// TIA Portal V16 export
// export: Created 2020-03-17T19:47:24.6378532Z, ExportSetting None, DisplayName Totally Integrated Automation Portal, DisplayVersion V16, DisplayName TIA Portal Version Control Interface, DisplayVersion V16, DisplayName TIA Portal Openness, DisplayVersion V16, DisplayName STEP 7 Professional, DisplayVersion V16, DisplayName STEP 7 Safety, DisplayVersion V16, DisplayName WinCC Advanced, DisplayVersion V16
FUNCTION_BLOCK "FB_R134a_BU_Valves"   // FB1303, LAD
TITLE = Base unit valve control // Grundeinheit Ventilsteuerung
{ S7_Optimized_Access := 'TRUE' }
// stored: AutoNumber false, MemoryReserve 100, SetENOAutomatically false
   VAR
      Stat_Flag : Array[1..32] of Bool;   // Bits for edge detection // Bits für Flankenerkennung
      Valve_10 : "FB_VALVE";
      Valve_12 : "FB_VALVE";
      Valve_13 : "FB_VALVE";
      Valve_16 : "FB_VALVE";
      Valve_17 : "FB_VALVE";
      Valve_18 : "FB_VALVE";
      Valve_19 : "FB_VALVE";
      Valve_20 : "FB_VALVE";
      Valve_21 : "FB_VALVE";
      Valve_23 : "FB_VALVE";
      Valve_24 : "FB_VALVE";
      Valve_31 : "FB_VALVE";
      Valve_43 : "FB_VALVE";
      Valve_44 : "FB_VALVE";
      Valve_Spare_1 : "FB_VALVE";
      Valve_Spare_2 : "FB_VALVE";
      Valve_Spare_3 : "FB_VALVE";
      Valve_Spare_4 : "FB_VALVE";
      Valve_Spare_5 : "FB_VALVE";
      Valve_Spare_6 : "FB_VALVE";
   END_VAR
   VAR_TEMP
      Tmp_EnableMonitoring : Bool;   // Local monitoring release // Lokale Überwachungsfreigabe
      Tmp_EnableOperation : Bool;   // Local operation release // Lokale Startfreigabe
      Tmp_Bool : Bool;   // Placeholder BOOL // Platzhalter BOOL
      Tmp_Word : Word;   // Placeholder WORD // Platzhalter WORD
      Tmp_Int : Int;   // Placeholder INT // Platzhalter INT
      Tmp_Alarm : Array[1..4] of Bool;   // Temp variable for FB_Alarm // Temporäre Variablen für den FB_Alarm
      Tmp_CollectedAlarm : Bool;   // Temp collected alarm for FB_Alarm // Temporärer Sammelfehler für FB_Alarm
      Tmp_OffsetPropValveAir : Int;   // Offset value for proportional valve // Offsetwert für Proportionalventil
      Tmp_OffsetPropValveFluid : Int;   // Offset value for proportional valve // Offsetwert für Proportionalventil
      Tmp_Fault : Bool;   // Temp variable for fault // Temporäre Variable für Fehler
      Tmp_BypassRelivePressure : Bool;   // Bypass for function relive pressure // Beipass für die Funktion Druck entlasten
      Tmp_ReturnValue : Word;   // Return value from function // Rückgabewert von Funktion
   END_VAR
   VAR_TEMP   // added for the SCL form of the ladder/FBD networks
      _w1 : Bool;
   END_VAR
BEGIN

REGION Network 1: Enable Monitoring // Freigabe Überwachung
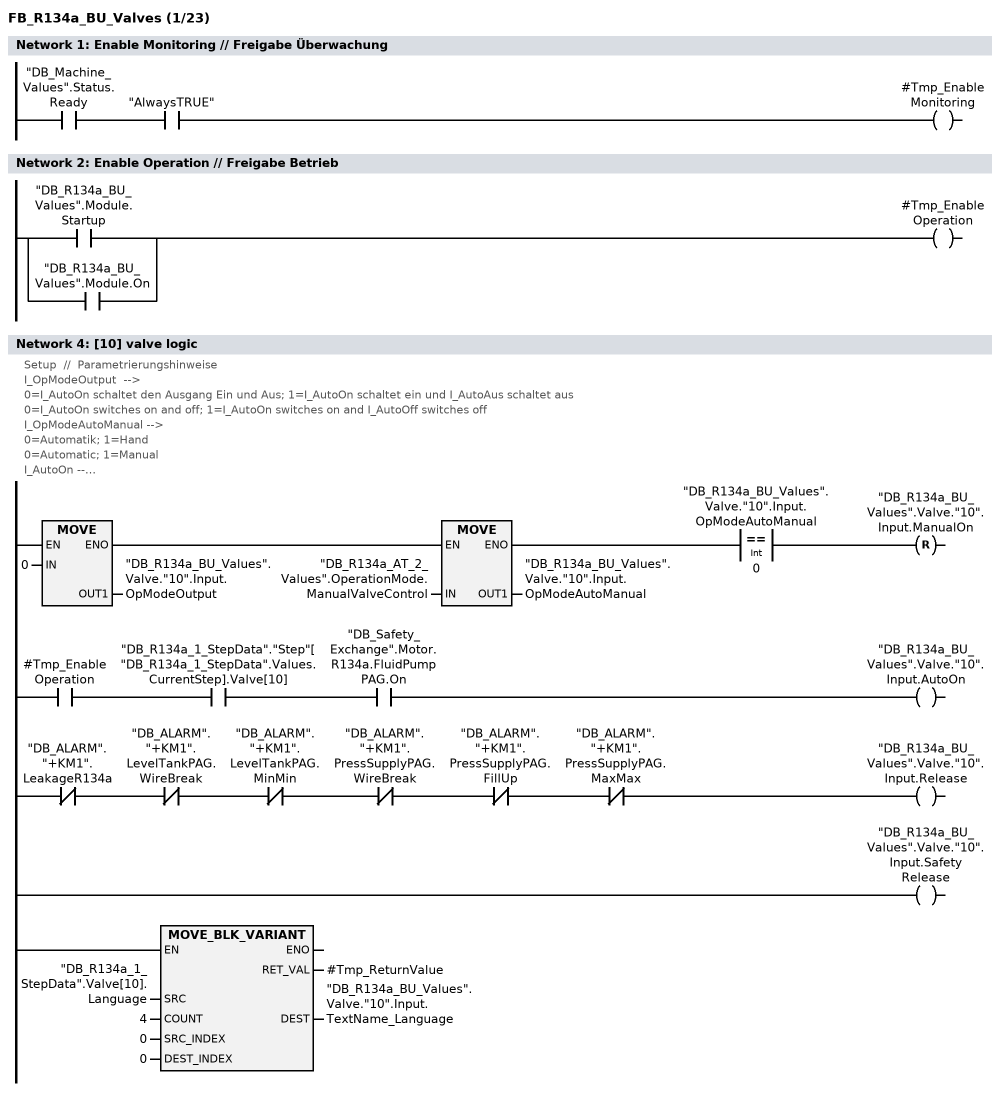
   RUNG wire#powerrail
      Contact( "DB_Machine_Values".Status.Ready )
      Contact( "AlwaysTRUE" )
      Coil( #Tmp_EnableMonitoring )
   END_RUNG
   // the same network as SCL:
   #Tmp_EnableMonitoring := "DB_Machine_Values".Status.Ready AND "AlwaysTRUE";
END_REGION

REGION Network 2: Enable Operation // Freigabe Betrieb
   RUNG wire#powerrail
      Contact( "DB_R134a_BU_Values".Module.Startup )
      wire#w1
      Coil( #Tmp_EnableOperation )
   END_RUNG
   RUNG wire#powerrail
      Contact( "DB_R134a_BU_Values".Module.On )
   END_RUNG wire#w1
   // the same network as SCL:
   #Tmp_EnableOperation := "DB_R134a_BU_Values".Module.Startup OR "DB_R134a_BU_Values".Module.On;
END_REGION

REGION Network 3: ------------- Valves base unit -------------
   // This network is only here to make the PLC program more structured/readable // Dieses Netzwerk ist nur hier um die Lesbarkeit des SPS-Programms zu erhöhen
END_REGION

REGION Network 4: [10] valve logic
   // Setup  //  Parametrierungshinweise
   // I_OpModeOutput  -->
   // 0=I_AutoOn schaltet den Ausgang Ein und Aus; 1=I_AutoOn schaltet ein und I_AutoAus schaltet aus
   // 0=I_AutoOn switches on and off; 1=I_AutoOn switches on and I_AutoOff switches off
   // 
   // I_OpModeAutoManual -->
   // 0=Automatik; 1=Hand
   // 0=Automatic; 1=Manual
   // 
   // I_AutoOn -->
   // 1=Automatik Ein, Eingang für die normalen Ventilverschaltungsbedingungen
   // 1=Automatic On, Input for the normal valve conditions
   // 
   // I_Release -->
   // 1=Freigabe, Eingang für die Fehlerbedingungen
   // 1=Release, Input for fault conditions
   // 
   // I_SafetyRelease -->
   // 1=Sicherheitsfreigabe, Eingang für zusätzliche Schaltbefehle aus dem Sicherheitsprogramm
   // 1=Safety release, Input for additional safety conditions from the safety program
   RUNG wire#powerrail
      Move(in := 0, out1 => "DB_R134a_BU_Values".Valve."10".Input.OpModeOutput)
      Move(in := "DB_R134a_AT_2_Values".OperationMode.ManualValveControl, out1 => "DB_R134a_BU_Values".Valve."10".Input.OpModeAutoManual)
      { S7_Templates := "SrcType := Int" } EQ_Contact(in1 := "DB_R134a_BU_Values".Valve."10".Input.OpModeAutoManual, in2 := 0)
      R_Coil( "DB_R134a_BU_Values".Valve."10".Input.ManualOn )
   END_RUNG
   RUNG wire#powerrail
      Contact( #Tmp_EnableOperation )
      Contact( "DB_R134a_1_StepData"."Step"["DB_R134a_1_StepData".Values.CurrentStep].Valve[10] )
      Contact( "DB_Safety_Exchange".Motor.R134a.FluidPumpPAG.On )
      Coil( "DB_R134a_BU_Values".Valve."10".Input.AutoOn )
   END_RUNG
   RUNG wire#powerrail
      I_Contact( "DB_ALARM"."+KM1".LeakageR134a )
      I_Contact( "DB_ALARM"."+KM1".LevelTankPAG.WireBreak )
      I_Contact( "DB_ALARM"."+KM1".LevelTankPAG.MinMin )
      I_Contact( "DB_ALARM"."+KM1".PressSupplyPAG.WireBreak )
      I_Contact( "DB_ALARM"."+KM1".PressSupplyPAG.FillUp )
      I_Contact( "DB_ALARM"."+KM1".PressSupplyPAG.MaxMax )
      Coil( "DB_R134a_BU_Values".Valve."10".Input.Release )
   END_RUNG
   RUNG wire#powerrail
      Coil( "DB_R134a_BU_Values".Valve."10".Input.SafetyRelease )
   END_RUNG
   RUNG wire#powerrail
      MOVE_BLK_VARIANT(SRC := "DB_R134a_1_StepData".Valve[10].Language, COUNT := 4, SRC_INDEX := 0, DEST_INDEX := 0, Ret_Val => #Tmp_ReturnValue, DEST => "DB_R134a_BU_Values".Valve."10".Input.TextName_Language)
   END_RUNG
   // the same network as SCL:
   "DB_R134a_BU_Values".Valve."10".Input.OpModeOutput := 0;
   "DB_R134a_BU_Values".Valve."10".Input.OpModeAutoManual := "DB_R134a_AT_2_Values".OperationMode.ManualValveControl;
   IF "DB_R134a_BU_Values".Valve."10".Input.OpModeAutoManual = 0 THEN
       "DB_R134a_BU_Values".Valve."10".Input.ManualOn := FALSE;
   END_IF;
   "DB_R134a_BU_Values".Valve."10".Input.AutoOn := #Tmp_EnableOperation AND "DB_R134a_1_StepData"."Step"["DB_R134a_1_StepData".Values.CurrentStep].Valve[10] AND "DB_Safety_Exchange".Motor.R134a.FluidPumpPAG.On;
   "DB_R134a_BU_Values".Valve."10".Input.Release := NOT "DB_ALARM"."+KM1".LeakageR134a AND NOT "DB_ALARM"."+KM1".LevelTankPAG.WireBreak AND NOT "DB_ALARM"."+KM1".LevelTankPAG.MinMin AND NOT "DB_ALARM"."+KM1".PressSupplyPAG.WireBreak AND NOT "DB_ALARM"."+KM1".PressSupplyPAG.FillUp AND NOT "DB_ALARM"."+KM1".PressSupplyPAG.MaxMax;
   "DB_R134a_BU_Values".Valve."10".Input.SafetyRelease := TRUE;
   #Tmp_ReturnValue := MOVE_BLK_VARIANT(SRC := "DB_R134a_1_StepData".Valve[10].Language,
                           COUNT := 4,
                           SRC_INDEX := 0,
                           DEST_INDEX := 0,
                           DEST => "DB_R134a_BU_Values".Valve."10".Input.TextName_Language);
END_REGION

REGION Network 5: [10] valve 1KM1VI1KKP9KK101 - 100.101.6 - Charge accumulator PAG // Füllen PAG-Speicher
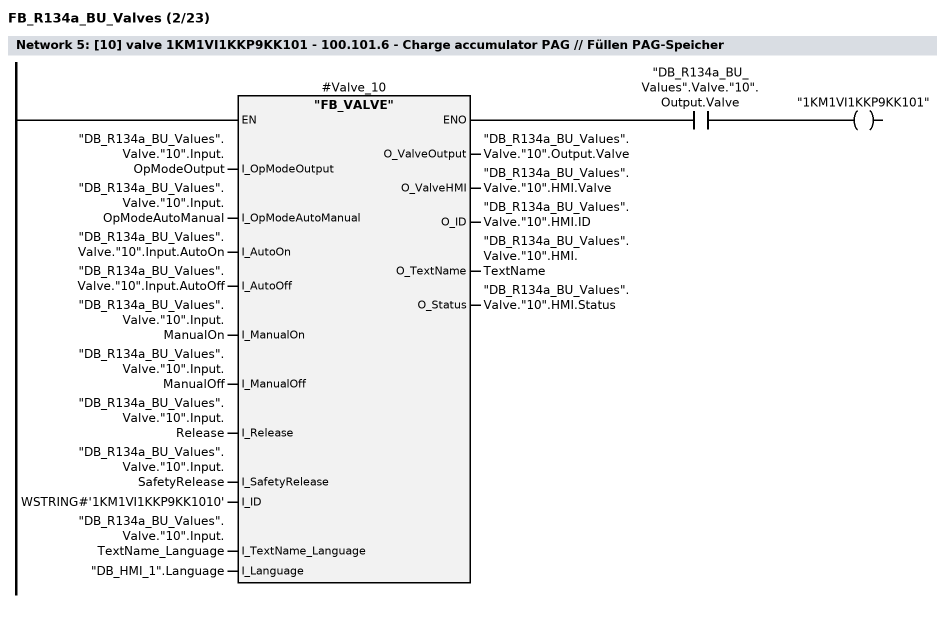
   RUNG wire#powerrail
      #Valve_10(I_OpModeOutput := "DB_R134a_BU_Values".Valve."10".Input.OpModeOutput, I_OpModeAutoManual := "DB_R134a_BU_Values".Valve."10".Input.OpModeAutoManual, I_AutoOn := "DB_R134a_BU_Values".Valve."10".Input.AutoOn, I_AutoOff := "DB_R134a_BU_Values".Valve."10".Input.AutoOff, I_ManualOn := "DB_R134a_BU_Values".Valve."10".Input.ManualOn, I_ManualOff := "DB_R134a_BU_Values".Valve."10".Input.ManualOff, I_Release := "DB_R134a_BU_Values".Valve."10".Input.Release, I_SafetyRelease := "DB_R134a_BU_Values".Valve."10".Input.SafetyRelease, I_ID := WSTRING#'1KM1VI1KKP9KK1010', I_TextName_Language := "DB_R134a_BU_Values".Valve."10".Input.TextName_Language, I_Language := "DB_HMI_1".Language, O_ValveOutput => "DB_R134a_BU_Values".Valve."10".Output.Valve, O_ValveHMI => "DB_R134a_BU_Values".Valve."10".HMI.Valve, O_ID => "DB_R134a_BU_Values".Valve."10".HMI.ID, O_TextName => "DB_R134a_BU_Values".Valve."10".HMI.TextName, O_Status => "DB_R134a_BU_Values".Valve."10".HMI.Status)
      Contact( "DB_R134a_BU_Values".Valve."10".Output.Valve )
      Coil( "1KM1VI1KKP9KK101" )
   END_RUNG
   // the same network as SCL:
   #Valve_10(I_OpModeOutput := "DB_R134a_BU_Values".Valve."10".Input.OpModeOutput,   // "FB_VALVE"
             I_OpModeAutoManual := "DB_R134a_BU_Values".Valve."10".Input.OpModeAutoManual,
             I_AutoOn := "DB_R134a_BU_Values".Valve."10".Input.AutoOn,
             I_AutoOff := "DB_R134a_BU_Values".Valve."10".Input.AutoOff,
             I_ManualOn := "DB_R134a_BU_Values".Valve."10".Input.ManualOn,
             I_ManualOff := "DB_R134a_BU_Values".Valve."10".Input.ManualOff,
             I_Release := "DB_R134a_BU_Values".Valve."10".Input.Release,
             I_SafetyRelease := "DB_R134a_BU_Values".Valve."10".Input.SafetyRelease,
             I_ID := WSTRING#'1KM1VI1KKP9KK1010',
             I_TextName_Language := "DB_R134a_BU_Values".Valve."10".Input.TextName_Language,
             I_Language := "DB_HMI_1".Language,
             O_ValveOutput => "DB_R134a_BU_Values".Valve."10".Output.Valve,
             O_ValveHMI => "DB_R134a_BU_Values".Valve."10".HMI.Valve,
             O_ID => "DB_R134a_BU_Values".Valve."10".HMI.ID,
             O_TextName => "DB_R134a_BU_Values".Valve."10".HMI.TextName,
             O_Status => "DB_R134a_BU_Values".Valve."10".HMI.Status,
             ENO => #_w1);
   "1KM1VI1KKP9KK101" := #_w1 AND "DB_R134a_BU_Values".Valve."10".Output.Valve;
END_REGION

REGION Network 6: [12] valve logic
   // Setup  //  Parametrierungshinweise
   // I_OpModeOutput  -->
   // 0=I_AutoOn schaltet den Ausgang Ein und Aus; 1=I_AutoOn schaltet ein und I_AutoAus schaltet aus
   // 0=I_AutoOn switches on and off; 1=I_AutoOn switches on and I_AutoOff switches off
   // 
   // I_OpModeAutoManual -->
   // 0=Automatik; 1=Hand
   // 0=Automatic; 1=Manual
   // 
   // I_AutoOn -->
   // 1=Automatik Ein, Eingang für die normalen Ventilverschaltungsbedingungen
   // 1=Automatic On, Input for the normal valve conditions
   // 
   // I_Release -->
   // 1=Freigabe, Eingang für die Fehlerbedingungen
   // 1=Release, Input for fault conditions
   // 
   // I_SafetyRelease -->
   // 1=Sicherheitsfreigabe, Eingang für zusätzliche Schaltbefehle aus dem Sicherheitsprogramm
   // 1=Safety release, Input for additional safety conditions from the safety program
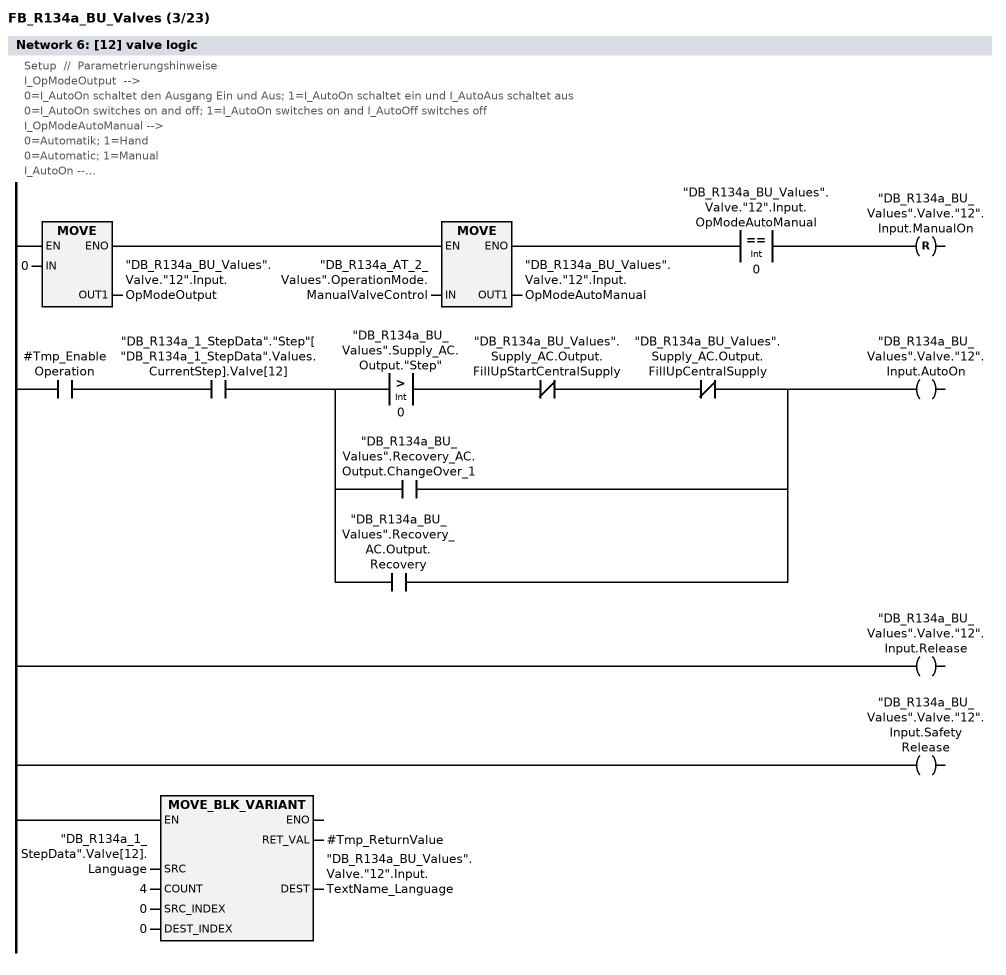
   RUNG wire#powerrail
      Move(in := 0, out1 => "DB_R134a_BU_Values".Valve."12".Input.OpModeOutput)
      Move(in := "DB_R134a_AT_2_Values".OperationMode.ManualValveControl, out1 => "DB_R134a_BU_Values".Valve."12".Input.OpModeAutoManual)
      { S7_Templates := "SrcType := Int" } EQ_Contact(in1 := "DB_R134a_BU_Values".Valve."12".Input.OpModeAutoManual, in2 := 0)
      R_Coil( "DB_R134a_BU_Values".Valve."12".Input.ManualOn )
   END_RUNG
   RUNG wire#powerrail
      Contact( #Tmp_EnableOperation )
      Contact( "DB_R134a_1_StepData"."Step"["DB_R134a_1_StepData".Values.CurrentStep].Valve[12] )
      wire#w1
      { S7_Templates := "SrcType := Int" } GT_Contact(in1 := "DB_R134a_BU_Values".Supply_AC.Output."Step", in2 := 0)
      I_Contact( "DB_R134a_BU_Values".Supply_AC.Output.FillUpStartCentralSupply )
      I_Contact( "DB_R134a_BU_Values".Supply_AC.Output.FillUpCentralSupply )
      wire#w2
      Coil( "DB_R134a_BU_Values".Valve."12".Input.AutoOn )
   END_RUNG
   RUNG wire#w1
      Contact( "DB_R134a_BU_Values".Recovery_AC.Output.ChangeOver_1 )
   END_RUNG wire#w2
   RUNG wire#w1
      Contact( "DB_R134a_BU_Values".Recovery_AC.Output.Recovery )
   END_RUNG wire#w2
   RUNG wire#powerrail
      Coil( "DB_R134a_BU_Values".Valve."12".Input.Release )
   END_RUNG
   RUNG wire#powerrail
      Coil( "DB_R134a_BU_Values".Valve."12".Input.SafetyRelease )
   END_RUNG
   RUNG wire#powerrail
      MOVE_BLK_VARIANT(SRC := "DB_R134a_1_StepData".Valve[12].Language, COUNT := 4, SRC_INDEX := 0, DEST_INDEX := 0, Ret_Val => #Tmp_ReturnValue, DEST => "DB_R134a_BU_Values".Valve."12".Input.TextName_Language)
   END_RUNG
   // the same network as SCL:
   "DB_R134a_BU_Values".Valve."12".Input.OpModeOutput := 0;
   "DB_R134a_BU_Values".Valve."12".Input.OpModeAutoManual := "DB_R134a_AT_2_Values".OperationMode.ManualValveControl;
   IF "DB_R134a_BU_Values".Valve."12".Input.OpModeAutoManual = 0 THEN
       "DB_R134a_BU_Values".Valve."12".Input.ManualOn := FALSE;
   END_IF;
   "DB_R134a_BU_Values".Valve."12".Input.AutoOn := #Tmp_EnableOperation AND "DB_R134a_1_StepData"."Step"["DB_R134a_1_StepData".Values.CurrentStep].Valve[12] AND ((("DB_R134a_BU_Values".Supply_AC.Output."Step" > 0) AND NOT "DB_R134a_BU_Values".Supply_AC.Output.FillUpStartCentralSupply AND NOT "DB_R134a_BU_Values".Supply_AC.Output.FillUpCentralSupply) OR "DB_R134a_BU_Values".Recovery_AC.Output.ChangeOver_1 OR "DB_R134a_BU_Values".Recovery_AC.Output.Recovery);
   "DB_R134a_BU_Values".Valve."12".Input.Release := TRUE;
   "DB_R134a_BU_Values".Valve."12".Input.SafetyRelease := TRUE;
   #Tmp_ReturnValue := MOVE_BLK_VARIANT(SRC := "DB_R134a_1_StepData".Valve[12].Language,
                           COUNT := 4,
                           SRC_INDEX := 0,
                           DEST_INDEX := 0,
                           DEST => "DB_R134a_BU_Values".Valve."12".Input.TextName_Language);
END_REGION

REGION Network 7: [12] valve 1KM1VI1KKP5KK420 - 109.420.3 - Compressed air supply (pump) // Druckluft Pumpe
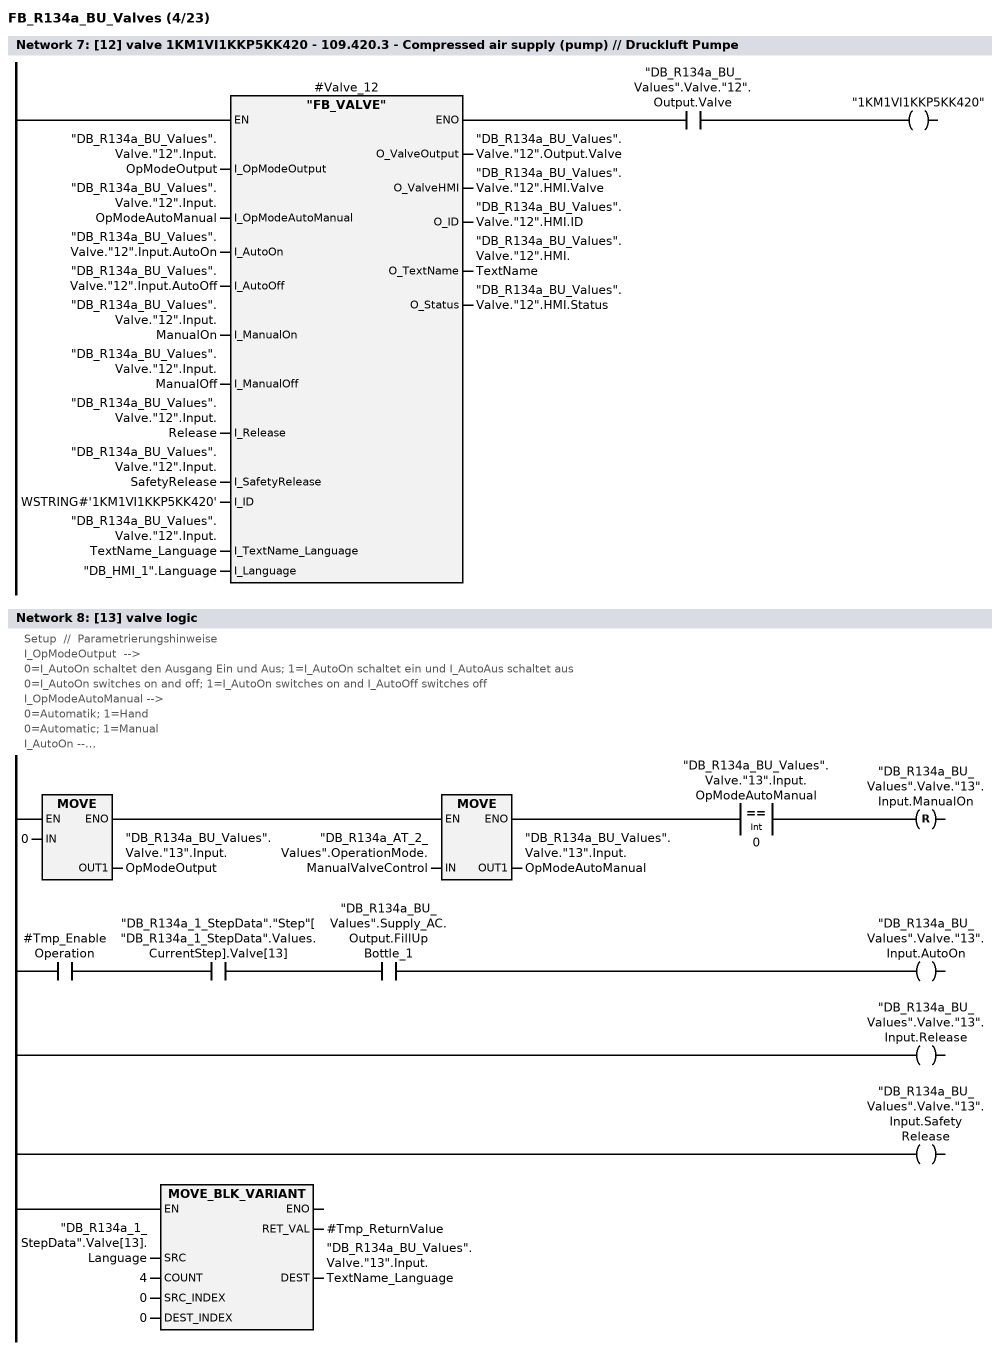
   RUNG wire#powerrail
      #Valve_12(I_OpModeOutput := "DB_R134a_BU_Values".Valve."12".Input.OpModeOutput, I_OpModeAutoManual := "DB_R134a_BU_Values".Valve."12".Input.OpModeAutoManual, I_AutoOn := "DB_R134a_BU_Values".Valve."12".Input.AutoOn, I_AutoOff := "DB_R134a_BU_Values".Valve."12".Input.AutoOff, I_ManualOn := "DB_R134a_BU_Values".Valve."12".Input.ManualOn, I_ManualOff := "DB_R134a_BU_Values".Valve."12".Input.ManualOff, I_Release := "DB_R134a_BU_Values".Valve."12".Input.Release, I_SafetyRelease := "DB_R134a_BU_Values".Valve."12".Input.SafetyRelease, I_ID := WSTRING#'1KM1VI1KKP5KK420', I_TextName_Language := "DB_R134a_BU_Values".Valve."12".Input.TextName_Language, I_Language := "DB_HMI_1".Language, O_ValveOutput => "DB_R134a_BU_Values".Valve."12".Output.Valve, O_ValveHMI => "DB_R134a_BU_Values".Valve."12".HMI.Valve, O_ID => "DB_R134a_BU_Values".Valve."12".HMI.ID, O_TextName => "DB_R134a_BU_Values".Valve."12".HMI.TextName, O_Status => "DB_R134a_BU_Values".Valve."12".HMI.Status)
      Contact( "DB_R134a_BU_Values".Valve."12".Output.Valve )
      Coil( "1KM1VI1KKP5KK420" )
   END_RUNG
   // the same network as SCL:
   #Valve_12(I_OpModeOutput := "DB_R134a_BU_Values".Valve."12".Input.OpModeOutput,   // "FB_VALVE"
             I_OpModeAutoManual := "DB_R134a_BU_Values".Valve."12".Input.OpModeAutoManual,
             I_AutoOn := "DB_R134a_BU_Values".Valve."12".Input.AutoOn,
             I_AutoOff := "DB_R134a_BU_Values".Valve."12".Input.AutoOff,
             I_ManualOn := "DB_R134a_BU_Values".Valve."12".Input.ManualOn,
             I_ManualOff := "DB_R134a_BU_Values".Valve."12".Input.ManualOff,
             I_Release := "DB_R134a_BU_Values".Valve."12".Input.Release,
             I_SafetyRelease := "DB_R134a_BU_Values".Valve."12".Input.SafetyRelease,
             I_ID := WSTRING#'1KM1VI1KKP5KK420',
             I_TextName_Language := "DB_R134a_BU_Values".Valve."12".Input.TextName_Language,
             I_Language := "DB_HMI_1".Language,
             O_ValveOutput => "DB_R134a_BU_Values".Valve."12".Output.Valve,
             O_ValveHMI => "DB_R134a_BU_Values".Valve."12".HMI.Valve,
             O_ID => "DB_R134a_BU_Values".Valve."12".HMI.ID,
             O_TextName => "DB_R134a_BU_Values".Valve."12".HMI.TextName,
             O_Status => "DB_R134a_BU_Values".Valve."12".HMI.Status,
             ENO => #_w1);
   "1KM1VI1KKP5KK420" := #_w1 AND "DB_R134a_BU_Values".Valve."12".Output.Valve;
END_REGION

REGION Network 8: [13] valve logic
   // Setup  //  Parametrierungshinweise
   // I_OpModeOutput  -->
   // 0=I_AutoOn schaltet den Ausgang Ein und Aus; 1=I_AutoOn schaltet ein und I_AutoAus schaltet aus
   // 0=I_AutoOn switches on and off; 1=I_AutoOn switches on and I_AutoOff switches off
   // 
   // I_OpModeAutoManual -->
   // 0=Automatik; 1=Hand
   // 0=Automatic; 1=Manual
   // 
   // I_AutoOn -->
   // 1=Automatik Ein, Eingang für die normalen Ventilverschaltungsbedingungen
   // 1=Automatic On, Input for the normal valve conditions
   // 
   // I_Release -->
   // 1=Freigabe, Eingang für die Fehlerbedingungen
   // 1=Release, Input for fault conditions
   // 
   // I_SafetyRelease -->
   // 1=Sicherheitsfreigabe, Eingang für zusätzliche Schaltbefehle aus dem Sicherheitsprogramm
   // 1=Safety release, Input for additional safety conditions from the safety program
   RUNG wire#powerrail
      Move(in := 0, out1 => "DB_R134a_BU_Values".Valve."13".Input.OpModeOutput)
      Move(in := "DB_R134a_AT_2_Values".OperationMode.ManualValveControl, out1 => "DB_R134a_BU_Values".Valve."13".Input.OpModeAutoManual)
      { S7_Templates := "SrcType := Int" } EQ_Contact(in1 := "DB_R134a_BU_Values".Valve."13".Input.OpModeAutoManual, in2 := 0)
      R_Coil( "DB_R134a_BU_Values".Valve."13".Input.ManualOn )
   END_RUNG
   RUNG wire#powerrail
      Contact( #Tmp_EnableOperation )
      Contact( "DB_R134a_1_StepData"."Step"["DB_R134a_1_StepData".Values.CurrentStep].Valve[13] )
      Contact( "DB_R134a_BU_Values".Supply_AC.Output.FillUpBottle_1 )
      Coil( "DB_R134a_BU_Values".Valve."13".Input.AutoOn )
   END_RUNG
   RUNG wire#powerrail
      Coil( "DB_R134a_BU_Values".Valve."13".Input.Release )
   END_RUNG
   RUNG wire#powerrail
      Coil( "DB_R134a_BU_Values".Valve."13".Input.SafetyRelease )
   END_RUNG
   RUNG wire#powerrail
      MOVE_BLK_VARIANT(SRC := "DB_R134a_1_StepData".Valve[13].Language, COUNT := 4, SRC_INDEX := 0, DEST_INDEX := 0, Ret_Val => #Tmp_ReturnValue, DEST => "DB_R134a_BU_Values".Valve."13".Input.TextName_Language)
   END_RUNG
   // the same network as SCL:
   "DB_R134a_BU_Values".Valve."13".Input.OpModeOutput := 0;
   "DB_R134a_BU_Values".Valve."13".Input.OpModeAutoManual := "DB_R134a_AT_2_Values".OperationMode.ManualValveControl;
   IF "DB_R134a_BU_Values".Valve."13".Input.OpModeAutoManual = 0 THEN
       "DB_R134a_BU_Values".Valve."13".Input.ManualOn := FALSE;
   END_IF;
   "DB_R134a_BU_Values".Valve."13".Input.AutoOn := #Tmp_EnableOperation AND "DB_R134a_1_StepData"."Step"["DB_R134a_1_StepData".Values.CurrentStep].Valve[13] AND "DB_R134a_BU_Values".Supply_AC.Output.FillUpBottle_1;
   "DB_R134a_BU_Values".Valve."13".Input.Release := TRUE;
   "DB_R134a_BU_Values".Valve."13".Input.SafetyRelease := TRUE;
   #Tmp_ReturnValue := MOVE_BLK_VARIANT(SRC := "DB_R134a_1_StepData".Valve[13].Language,
                           COUNT := 4,
                           SRC_INDEX := 0,
                           DEST_INDEX := 0,
                           DEST => "DB_R134a_BU_Values".Valve."13".Input.TextName_Language);
END_REGION

REGION Network 9: [13] valve 1KM1VI1KKP3KK30 - 100.30.3 - Supply – Bottle 1 // Versorgung - Flasche 1
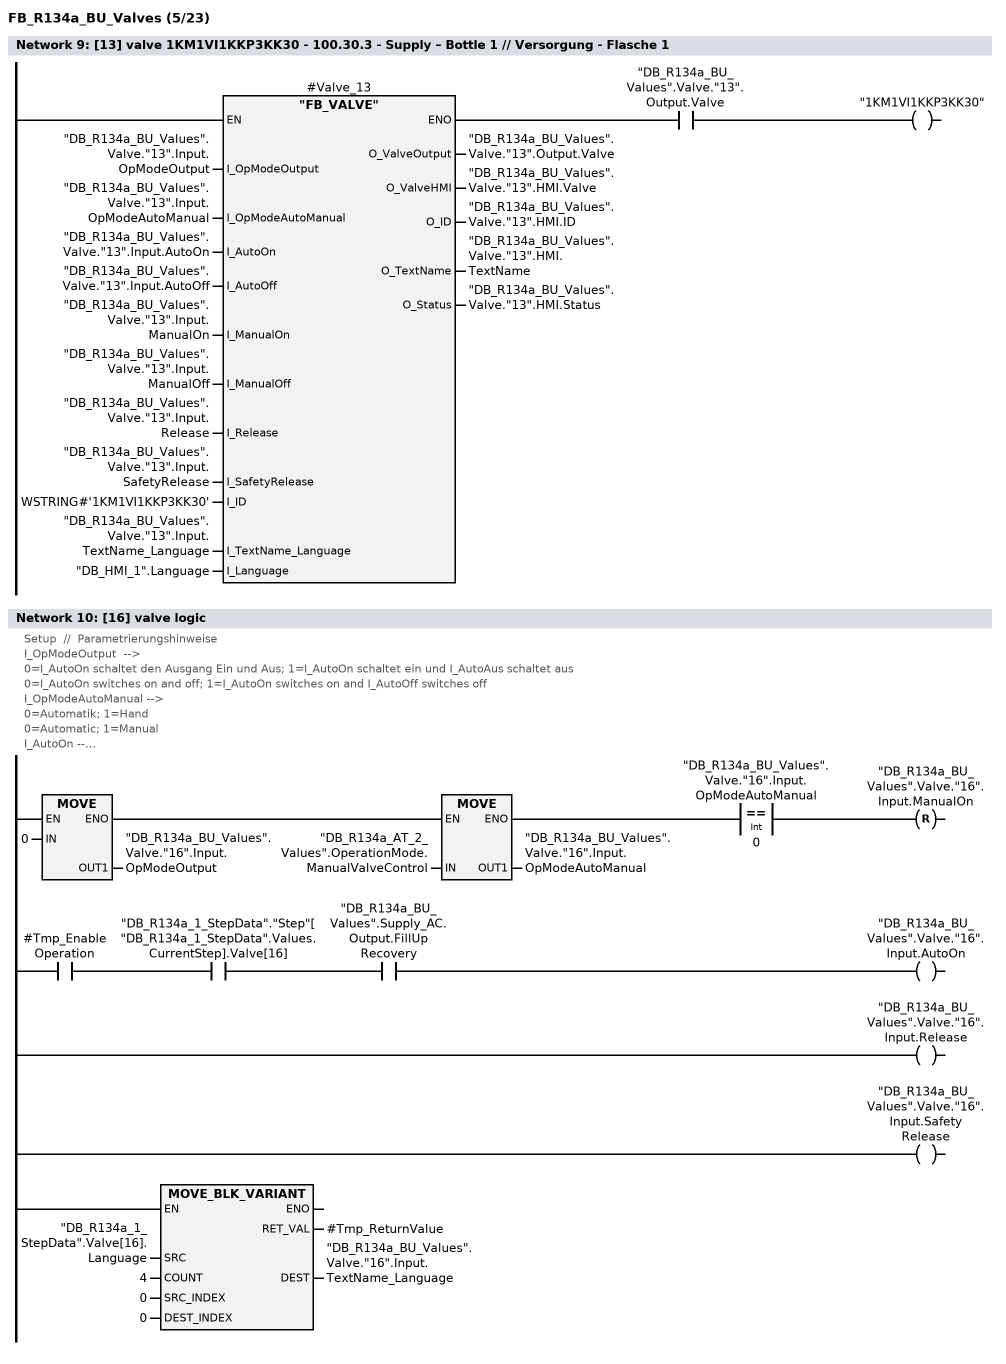
   RUNG wire#powerrail
      #Valve_13(I_OpModeOutput := "DB_R134a_BU_Values".Valve."13".Input.OpModeOutput, I_OpModeAutoManual := "DB_R134a_BU_Values".Valve."13".Input.OpModeAutoManual, I_AutoOn := "DB_R134a_BU_Values".Valve."13".Input.AutoOn, I_AutoOff := "DB_R134a_BU_Values".Valve."13".Input.AutoOff, I_ManualOn := "DB_R134a_BU_Values".Valve."13".Input.ManualOn, I_ManualOff := "DB_R134a_BU_Values".Valve."13".Input.ManualOff, I_Release := "DB_R134a_BU_Values".Valve."13".Input.Release, I_SafetyRelease := "DB_R134a_BU_Values".Valve."13".Input.SafetyRelease, I_ID := WSTRING#'1KM1VI1KKP3KK30', I_TextName_Language := "DB_R134a_BU_Values".Valve."13".Input.TextName_Language, I_Language := "DB_HMI_1".Language, O_ValveOutput => "DB_R134a_BU_Values".Valve."13".Output.Valve, O_ValveHMI => "DB_R134a_BU_Values".Valve."13".HMI.Valve, O_ID => "DB_R134a_BU_Values".Valve."13".HMI.ID, O_TextName => "DB_R134a_BU_Values".Valve."13".HMI.TextName, O_Status => "DB_R134a_BU_Values".Valve."13".HMI.Status)
      Contact( "DB_R134a_BU_Values".Valve."13".Output.Valve )
      Coil( "1KM1VI1KKP3KK30" )
   END_RUNG
   // the same network as SCL:
   #Valve_13(I_OpModeOutput := "DB_R134a_BU_Values".Valve."13".Input.OpModeOutput,   // "FB_VALVE"
             I_OpModeAutoManual := "DB_R134a_BU_Values".Valve."13".Input.OpModeAutoManual,
             I_AutoOn := "DB_R134a_BU_Values".Valve."13".Input.AutoOn,
             I_AutoOff := "DB_R134a_BU_Values".Valve."13".Input.AutoOff,
             I_ManualOn := "DB_R134a_BU_Values".Valve."13".Input.ManualOn,
             I_ManualOff := "DB_R134a_BU_Values".Valve."13".Input.ManualOff,
             I_Release := "DB_R134a_BU_Values".Valve."13".Input.Release,
             I_SafetyRelease := "DB_R134a_BU_Values".Valve."13".Input.SafetyRelease,
             I_ID := WSTRING#'1KM1VI1KKP3KK30',
             I_TextName_Language := "DB_R134a_BU_Values".Valve."13".Input.TextName_Language,
             I_Language := "DB_HMI_1".Language,
             O_ValveOutput => "DB_R134a_BU_Values".Valve."13".Output.Valve,
             O_ValveHMI => "DB_R134a_BU_Values".Valve."13".HMI.Valve,
             O_ID => "DB_R134a_BU_Values".Valve."13".HMI.ID,
             O_TextName => "DB_R134a_BU_Values".Valve."13".HMI.TextName,
             O_Status => "DB_R134a_BU_Values".Valve."13".HMI.Status,
             ENO => #_w1);
   "1KM1VI1KKP3KK30" := #_w1 AND "DB_R134a_BU_Values".Valve."13".Output.Valve;
END_REGION

REGION Network 10: [16] valve logic
   // Setup  //  Parametrierungshinweise
   // I_OpModeOutput  -->
   // 0=I_AutoOn schaltet den Ausgang Ein und Aus; 1=I_AutoOn schaltet ein und I_AutoAus schaltet aus
   // 0=I_AutoOn switches on and off; 1=I_AutoOn switches on and I_AutoOff switches off
   // 
   // I_OpModeAutoManual -->
   // 0=Automatik; 1=Hand
   // 0=Automatic; 1=Manual
   // 
   // I_AutoOn -->
   // 1=Automatik Ein, Eingang für die normalen Ventilverschaltungsbedingungen
   // 1=Automatic On, Input for the normal valve conditions
   // 
   // I_Release -->
   // 1=Freigabe, Eingang für die Fehlerbedingungen
   // 1=Release, Input for fault conditions
   // 
   // I_SafetyRelease -->
   // 1=Sicherheitsfreigabe, Eingang für zusätzliche Schaltbefehle aus dem Sicherheitsprogramm
   // 1=Safety release, Input for additional safety conditions from the safety program
   RUNG wire#powerrail
      Move(in := 0, out1 => "DB_R134a_BU_Values".Valve."16".Input.OpModeOutput)
      Move(in := "DB_R134a_AT_2_Values".OperationMode.ManualValveControl, out1 => "DB_R134a_BU_Values".Valve."16".Input.OpModeAutoManual)
      { S7_Templates := "SrcType := Int" } EQ_Contact(in1 := "DB_R134a_BU_Values".Valve."16".Input.OpModeAutoManual, in2 := 0)
      R_Coil( "DB_R134a_BU_Values".Valve."16".Input.ManualOn )
   END_RUNG
   RUNG wire#powerrail
      Contact( #Tmp_EnableOperation )
      Contact( "DB_R134a_1_StepData"."Step"["DB_R134a_1_StepData".Values.CurrentStep].Valve[16] )
      Contact( "DB_R134a_BU_Values".Supply_AC.Output.FillUpRecovery )
      Coil( "DB_R134a_BU_Values".Valve."16".Input.AutoOn )
   END_RUNG
   RUNG wire#powerrail
      Coil( "DB_R134a_BU_Values".Valve."16".Input.Release )
   END_RUNG
   RUNG wire#powerrail
      Coil( "DB_R134a_BU_Values".Valve."16".Input.SafetyRelease )
   END_RUNG
   RUNG wire#powerrail
      MOVE_BLK_VARIANT(SRC := "DB_R134a_1_StepData".Valve[16].Language, COUNT := 4, SRC_INDEX := 0, DEST_INDEX := 0, Ret_Val => #Tmp_ReturnValue, DEST => "DB_R134a_BU_Values".Valve."16".Input.TextName_Language)
   END_RUNG
   // the same network as SCL:
   "DB_R134a_BU_Values".Valve."16".Input.OpModeOutput := 0;
   "DB_R134a_BU_Values".Valve."16".Input.OpModeAutoManual := "DB_R134a_AT_2_Values".OperationMode.ManualValveControl;
   IF "DB_R134a_BU_Values".Valve."16".Input.OpModeAutoManual = 0 THEN
       "DB_R134a_BU_Values".Valve."16".Input.ManualOn := FALSE;
   END_IF;
   "DB_R134a_BU_Values".Valve."16".Input.AutoOn := #Tmp_EnableOperation AND "DB_R134a_1_StepData"."Step"["DB_R134a_1_StepData".Values.CurrentStep].Valve[16] AND "DB_R134a_BU_Values".Supply_AC.Output.FillUpRecovery;
   "DB_R134a_BU_Values".Valve."16".Input.Release := TRUE;
   "DB_R134a_BU_Values".Valve."16".Input.SafetyRelease := TRUE;
   #Tmp_ReturnValue := MOVE_BLK_VARIANT(SRC := "DB_R134a_1_StepData".Valve[16].Language,
                           COUNT := 4,
                           SRC_INDEX := 0,
                           DEST_INDEX := 0,
                           DEST => "DB_R134a_BU_Values".Valve."16".Input.TextName_Language);
END_REGION

REGION Network 11: [16] valve 1KM1VI1KKP3KK70 - 100.70.3 - Supply from recovery accumulator // Versorgung - aus Rücksaugebehälter
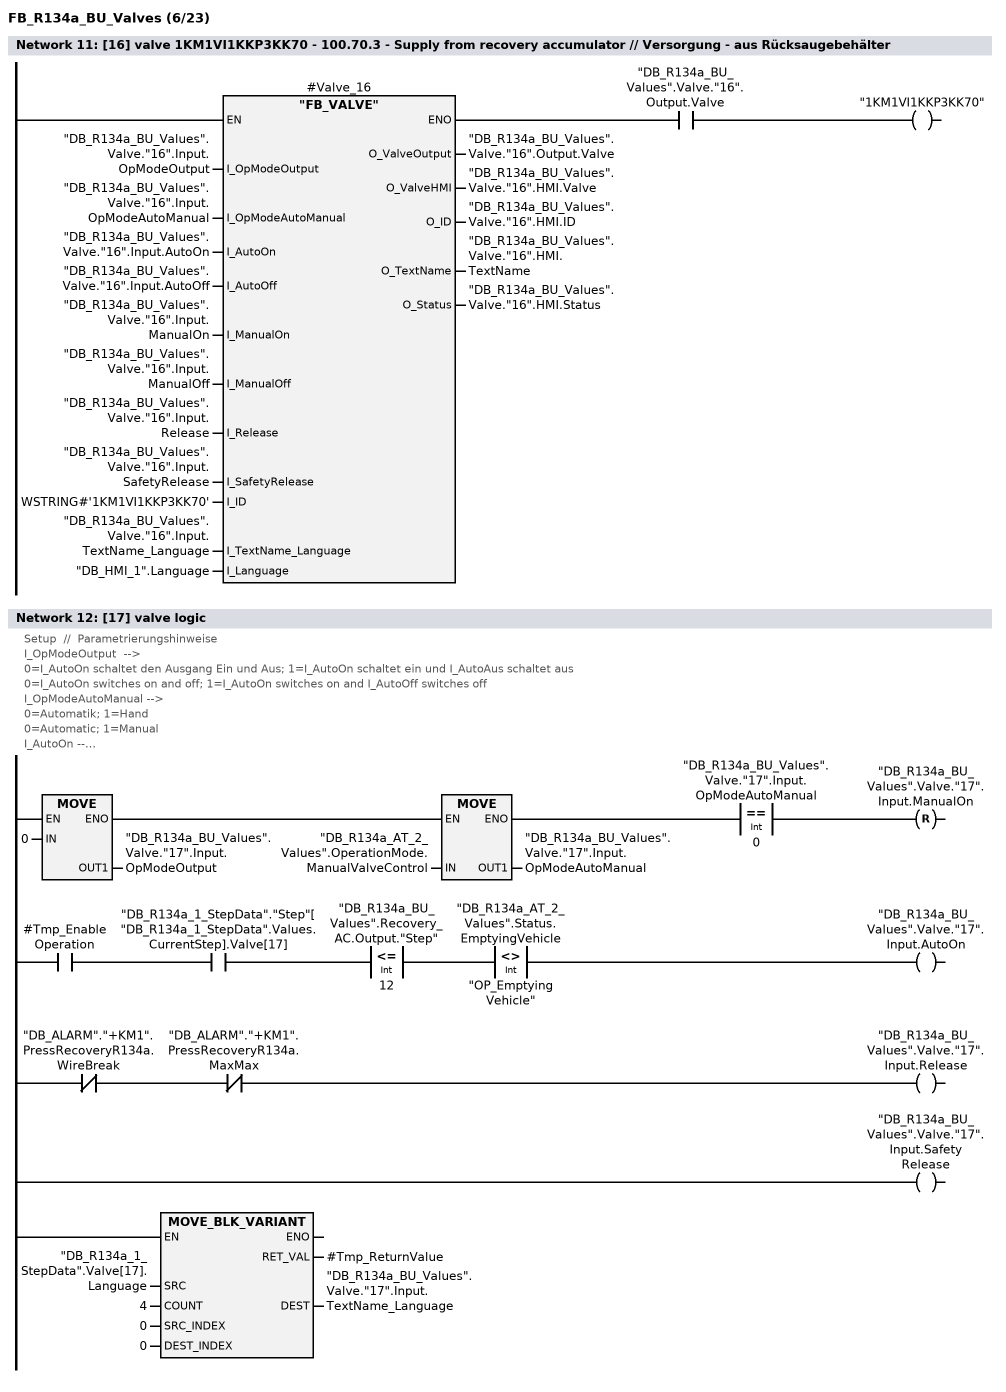
   RUNG wire#powerrail
      #Valve_16(I_OpModeOutput := "DB_R134a_BU_Values".Valve."16".Input.OpModeOutput, I_OpModeAutoManual := "DB_R134a_BU_Values".Valve."16".Input.OpModeAutoManual, I_AutoOn := "DB_R134a_BU_Values".Valve."16".Input.AutoOn, I_AutoOff := "DB_R134a_BU_Values".Valve."16".Input.AutoOff, I_ManualOn := "DB_R134a_BU_Values".Valve."16".Input.ManualOn, I_ManualOff := "DB_R134a_BU_Values".Valve."16".Input.ManualOff, I_Release := "DB_R134a_BU_Values".Valve."16".Input.Release, I_SafetyRelease := "DB_R134a_BU_Values".Valve."16".Input.SafetyRelease, I_ID := WSTRING#'1KM1VI1KKP3KK70', I_TextName_Language := "DB_R134a_BU_Values".Valve."16".Input.TextName_Language, I_Language := "DB_HMI_1".Language, O_ValveOutput => "DB_R134a_BU_Values".Valve."16".Output.Valve, O_ValveHMI => "DB_R134a_BU_Values".Valve."16".HMI.Valve, O_ID => "DB_R134a_BU_Values".Valve."16".HMI.ID, O_TextName => "DB_R134a_BU_Values".Valve."16".HMI.TextName, O_Status => "DB_R134a_BU_Values".Valve."16".HMI.Status)
      Contact( "DB_R134a_BU_Values".Valve."16".Output.Valve )
      Coil( "1KM1VI1KKP3KK70" )
   END_RUNG
   // the same network as SCL:
   #Valve_16(I_OpModeOutput := "DB_R134a_BU_Values".Valve."16".Input.OpModeOutput,   // "FB_VALVE"
             I_OpModeAutoManual := "DB_R134a_BU_Values".Valve."16".Input.OpModeAutoManual,
             I_AutoOn := "DB_R134a_BU_Values".Valve."16".Input.AutoOn,
             I_AutoOff := "DB_R134a_BU_Values".Valve."16".Input.AutoOff,
             I_ManualOn := "DB_R134a_BU_Values".Valve."16".Input.ManualOn,
             I_ManualOff := "DB_R134a_BU_Values".Valve."16".Input.ManualOff,
             I_Release := "DB_R134a_BU_Values".Valve."16".Input.Release,
             I_SafetyRelease := "DB_R134a_BU_Values".Valve."16".Input.SafetyRelease,
             I_ID := WSTRING#'1KM1VI1KKP3KK70',
             I_TextName_Language := "DB_R134a_BU_Values".Valve."16".Input.TextName_Language,
             I_Language := "DB_HMI_1".Language,
             O_ValveOutput => "DB_R134a_BU_Values".Valve."16".Output.Valve,
             O_ValveHMI => "DB_R134a_BU_Values".Valve."16".HMI.Valve,
             O_ID => "DB_R134a_BU_Values".Valve."16".HMI.ID,
             O_TextName => "DB_R134a_BU_Values".Valve."16".HMI.TextName,
             O_Status => "DB_R134a_BU_Values".Valve."16".HMI.Status,
             ENO => #_w1);
   "1KM1VI1KKP3KK70" := #_w1 AND "DB_R134a_BU_Values".Valve."16".Output.Valve;
END_REGION

REGION Network 12: [17] valve logic
   // Setup  //  Parametrierungshinweise
   // I_OpModeOutput  -->
   // 0=I_AutoOn schaltet den Ausgang Ein und Aus; 1=I_AutoOn schaltet ein und I_AutoAus schaltet aus
   // 0=I_AutoOn switches on and off; 1=I_AutoOn switches on and I_AutoOff switches off
   // 
   // I_OpModeAutoManual -->
   // 0=Automatik; 1=Hand
   // 0=Automatic; 1=Manual
   // 
   // I_AutoOn -->
   // 1=Automatik Ein, Eingang für die normalen Ventilverschaltungsbedingungen
   // 1=Automatic On, Input for the normal valve conditions
   // 
   // I_Release -->
   // 1=Freigabe, Eingang für die Fehlerbedingungen
   // 1=Release, Input for fault conditions
   // 
   // I_SafetyRelease -->
   // 1=Sicherheitsfreigabe, Eingang für zusätzliche Schaltbefehle aus dem Sicherheitsprogramm
   // 1=Safety release, Input for additional safety conditions from the safety program
   RUNG wire#powerrail
      Move(in := 0, out1 => "DB_R134a_BU_Values".Valve."17".Input.OpModeOutput)
      Move(in := "DB_R134a_AT_2_Values".OperationMode.ManualValveControl, out1 => "DB_R134a_BU_Values".Valve."17".Input.OpModeAutoManual)
      { S7_Templates := "SrcType := Int" } EQ_Contact(in1 := "DB_R134a_BU_Values".Valve."17".Input.OpModeAutoManual, in2 := 0)
      R_Coil( "DB_R134a_BU_Values".Valve."17".Input.ManualOn )
   END_RUNG
   RUNG wire#powerrail
      Contact( #Tmp_EnableOperation )
      Contact( "DB_R134a_1_StepData"."Step"["DB_R134a_1_StepData".Values.CurrentStep].Valve[17] )
      { S7_Templates := "SrcType := Int" } LE_Contact(in1 := "DB_R134a_BU_Values".Recovery_AC.Output."Step", in2 := 12)
      { S7_Templates := "SrcType := Int" } NE_Contact(in1 := "DB_R134a_AT_2_Values".Status.EmptyingVehicle, in2 := "OP_EmptyingVehicle")
      Coil( "DB_R134a_BU_Values".Valve."17".Input.AutoOn )
   END_RUNG
   RUNG wire#powerrail
      I_Contact( "DB_ALARM"."+KM1".PressRecoveryR134a.WireBreak )
      I_Contact( "DB_ALARM"."+KM1".PressRecoveryR134a.MaxMax )
      Coil( "DB_R134a_BU_Values".Valve."17".Input.Release )
   END_RUNG
   RUNG wire#powerrail
      Coil( "DB_R134a_BU_Values".Valve."17".Input.SafetyRelease )
   END_RUNG
   RUNG wire#powerrail
      MOVE_BLK_VARIANT(SRC := "DB_R134a_1_StepData".Valve[17].Language, COUNT := 4, SRC_INDEX := 0, DEST_INDEX := 0, Ret_Val => #Tmp_ReturnValue, DEST => "DB_R134a_BU_Values".Valve."17".Input.TextName_Language)
   END_RUNG
   // the same network as SCL:
   "DB_R134a_BU_Values".Valve."17".Input.OpModeOutput := 0;
   "DB_R134a_BU_Values".Valve."17".Input.OpModeAutoManual := "DB_R134a_AT_2_Values".OperationMode.ManualValveControl;
   IF "DB_R134a_BU_Values".Valve."17".Input.OpModeAutoManual = 0 THEN
       "DB_R134a_BU_Values".Valve."17".Input.ManualOn := FALSE;
   END_IF;
   "DB_R134a_BU_Values".Valve."17".Input.AutoOn := #Tmp_EnableOperation AND "DB_R134a_1_StepData"."Step"["DB_R134a_1_StepData".Values.CurrentStep].Valve[17] AND ("DB_R134a_BU_Values".Recovery_AC.Output."Step" <= 12) AND ("DB_R134a_AT_2_Values".Status.EmptyingVehicle <> "OP_EmptyingVehicle");
   "DB_R134a_BU_Values".Valve."17".Input.Release := NOT "DB_ALARM"."+KM1".PressRecoveryR134a.WireBreak AND NOT "DB_ALARM"."+KM1".PressRecoveryR134a.MaxMax;
   "DB_R134a_BU_Values".Valve."17".Input.SafetyRelease := TRUE;
   #Tmp_ReturnValue := MOVE_BLK_VARIANT(SRC := "DB_R134a_1_StepData".Valve[17].Language,
                           COUNT := 4,
                           SRC_INDEX := 0,
                           DEST_INDEX := 0,
                           DEST => "DB_R134a_BU_Values".Valve."17".Input.TextName_Language);
END_REGION

REGION Network 13: [17] valve 1KM1VI1KKP5KK384 - 100.384.3 - Recovery - Test bottle // Rückgewinnung - Flasche
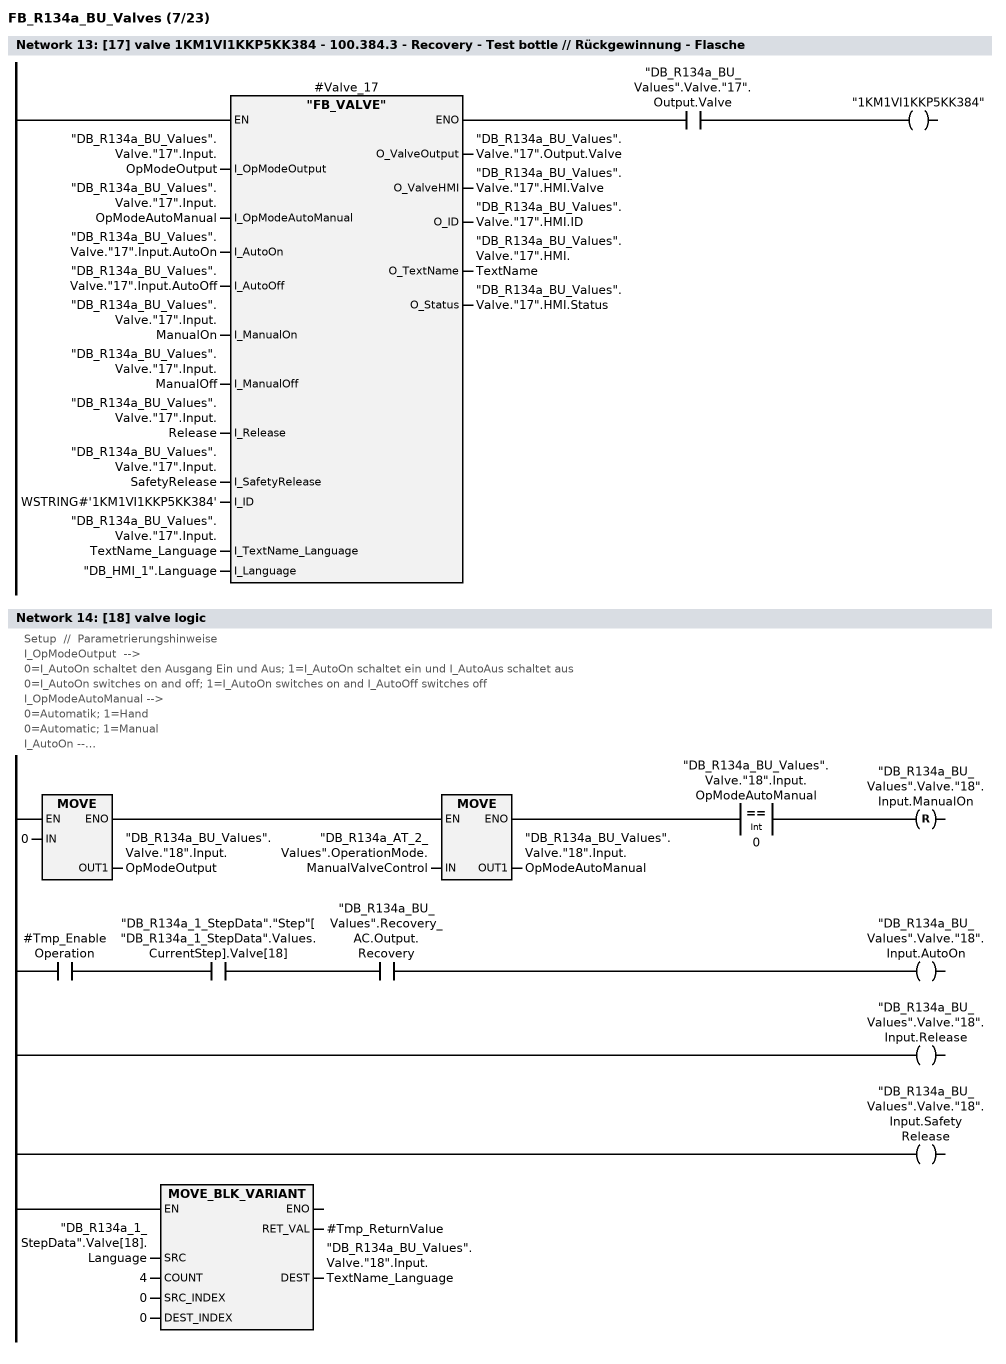
   RUNG wire#powerrail
      #Valve_17(I_OpModeOutput := "DB_R134a_BU_Values".Valve."17".Input.OpModeOutput, I_OpModeAutoManual := "DB_R134a_BU_Values".Valve."17".Input.OpModeAutoManual, I_AutoOn := "DB_R134a_BU_Values".Valve."17".Input.AutoOn, I_AutoOff := "DB_R134a_BU_Values".Valve."17".Input.AutoOff, I_ManualOn := "DB_R134a_BU_Values".Valve."17".Input.ManualOn, I_ManualOff := "DB_R134a_BU_Values".Valve."17".Input.ManualOff, I_Release := "DB_R134a_BU_Values".Valve."17".Input.Release, I_SafetyRelease := "DB_R134a_BU_Values".Valve."17".Input.SafetyRelease, I_ID := WSTRING#'1KM1VI1KKP5KK384', I_TextName_Language := "DB_R134a_BU_Values".Valve."17".Input.TextName_Language, I_Language := "DB_HMI_1".Language, O_ValveOutput => "DB_R134a_BU_Values".Valve."17".Output.Valve, O_ValveHMI => "DB_R134a_BU_Values".Valve."17".HMI.Valve, O_ID => "DB_R134a_BU_Values".Valve."17".HMI.ID, O_TextName => "DB_R134a_BU_Values".Valve."17".HMI.TextName, O_Status => "DB_R134a_BU_Values".Valve."17".HMI.Status)
      Contact( "DB_R134a_BU_Values".Valve."17".Output.Valve )
      Coil( "1KM1VI1KKP5KK384" )
   END_RUNG
   // the same network as SCL:
   #Valve_17(I_OpModeOutput := "DB_R134a_BU_Values".Valve."17".Input.OpModeOutput,   // "FB_VALVE"
             I_OpModeAutoManual := "DB_R134a_BU_Values".Valve."17".Input.OpModeAutoManual,
             I_AutoOn := "DB_R134a_BU_Values".Valve."17".Input.AutoOn,
             I_AutoOff := "DB_R134a_BU_Values".Valve."17".Input.AutoOff,
             I_ManualOn := "DB_R134a_BU_Values".Valve."17".Input.ManualOn,
             I_ManualOff := "DB_R134a_BU_Values".Valve."17".Input.ManualOff,
             I_Release := "DB_R134a_BU_Values".Valve."17".Input.Release,
             I_SafetyRelease := "DB_R134a_BU_Values".Valve."17".Input.SafetyRelease,
             I_ID := WSTRING#'1KM1VI1KKP5KK384',
             I_TextName_Language := "DB_R134a_BU_Values".Valve."17".Input.TextName_Language,
             I_Language := "DB_HMI_1".Language,
             O_ValveOutput => "DB_R134a_BU_Values".Valve."17".Output.Valve,
             O_ValveHMI => "DB_R134a_BU_Values".Valve."17".HMI.Valve,
             O_ID => "DB_R134a_BU_Values".Valve."17".HMI.ID,
             O_TextName => "DB_R134a_BU_Values".Valve."17".HMI.TextName,
             O_Status => "DB_R134a_BU_Values".Valve."17".HMI.Status,
             ENO => #_w1);
   "1KM1VI1KKP5KK384" := #_w1 AND "DB_R134a_BU_Values".Valve."17".Output.Valve;
END_REGION

REGION Network 14: [18] valve logic
   // Setup  //  Parametrierungshinweise
   // I_OpModeOutput  -->
   // 0=I_AutoOn schaltet den Ausgang Ein und Aus; 1=I_AutoOn schaltet ein und I_AutoAus schaltet aus
   // 0=I_AutoOn switches on and off; 1=I_AutoOn switches on and I_AutoOff switches off
   // 
   // I_OpModeAutoManual -->
   // 0=Automatik; 1=Hand
   // 0=Automatic; 1=Manual
   // 
   // I_AutoOn -->
   // 1=Automatik Ein, Eingang für die normalen Ventilverschaltungsbedingungen
   // 1=Automatic On, Input for the normal valve conditions
   // 
   // I_Release -->
   // 1=Freigabe, Eingang für die Fehlerbedingungen
   // 1=Release, Input for fault conditions
   // 
   // I_SafetyRelease -->
   // 1=Sicherheitsfreigabe, Eingang für zusätzliche Schaltbefehle aus dem Sicherheitsprogramm
   // 1=Safety release, Input for additional safety conditions from the safety program
   RUNG wire#powerrail
      Move(in := 0, out1 => "DB_R134a_BU_Values".Valve."18".Input.OpModeOutput)
      Move(in := "DB_R134a_AT_2_Values".OperationMode.ManualValveControl, out1 => "DB_R134a_BU_Values".Valve."18".Input.OpModeAutoManual)
      { S7_Templates := "SrcType := Int" } EQ_Contact(in1 := "DB_R134a_BU_Values".Valve."18".Input.OpModeAutoManual, in2 := 0)
      R_Coil( "DB_R134a_BU_Values".Valve."18".Input.ManualOn )
   END_RUNG
   RUNG wire#powerrail
      Contact( #Tmp_EnableOperation )
      Contact( "DB_R134a_1_StepData"."Step"["DB_R134a_1_StepData".Values.CurrentStep].Valve[18] )
      Contact( "DB_R134a_BU_Values".Recovery_AC.Output.Recovery )
      Coil( "DB_R134a_BU_Values".Valve."18".Input.AutoOn )
   END_RUNG
   RUNG wire#powerrail
      Coil( "DB_R134a_BU_Values".Valve."18".Input.Release )
   END_RUNG
   RUNG wire#powerrail
      Coil( "DB_R134a_BU_Values".Valve."18".Input.SafetyRelease )
   END_RUNG
   RUNG wire#powerrail
      MOVE_BLK_VARIANT(SRC := "DB_R134a_1_StepData".Valve[18].Language, COUNT := 4, SRC_INDEX := 0, DEST_INDEX := 0, Ret_Val => #Tmp_ReturnValue, DEST => "DB_R134a_BU_Values".Valve."18".Input.TextName_Language)
   END_RUNG
   // the same network as SCL:
   "DB_R134a_BU_Values".Valve."18".Input.OpModeOutput := 0;
   "DB_R134a_BU_Values".Valve."18".Input.OpModeAutoManual := "DB_R134a_AT_2_Values".OperationMode.ManualValveControl;
   IF "DB_R134a_BU_Values".Valve."18".Input.OpModeAutoManual = 0 THEN
       "DB_R134a_BU_Values".Valve."18".Input.ManualOn := FALSE;
   END_IF;
   "DB_R134a_BU_Values".Valve."18".Input.AutoOn := #Tmp_EnableOperation AND "DB_R134a_1_StepData"."Step"["DB_R134a_1_StepData".Values.CurrentStep].Valve[18] AND "DB_R134a_BU_Values".Recovery_AC.Output.Recovery;
   "DB_R134a_BU_Values".Valve."18".Input.Release := TRUE;
   "DB_R134a_BU_Values".Valve."18".Input.SafetyRelease := TRUE;
   #Tmp_ReturnValue := MOVE_BLK_VARIANT(SRC := "DB_R134a_1_StepData".Valve[18].Language,
                           COUNT := 4,
                           SRC_INDEX := 0,
                           DEST_INDEX := 0,
                           DEST => "DB_R134a_BU_Values".Valve."18".Input.TextName_Language);
END_REGION

REGION Network 15: [18] valve 1KM1VI1KKP4KK540 - 100.540.3 - Charge recovery tank // Auffüllen Rückgewinnungsbehälter
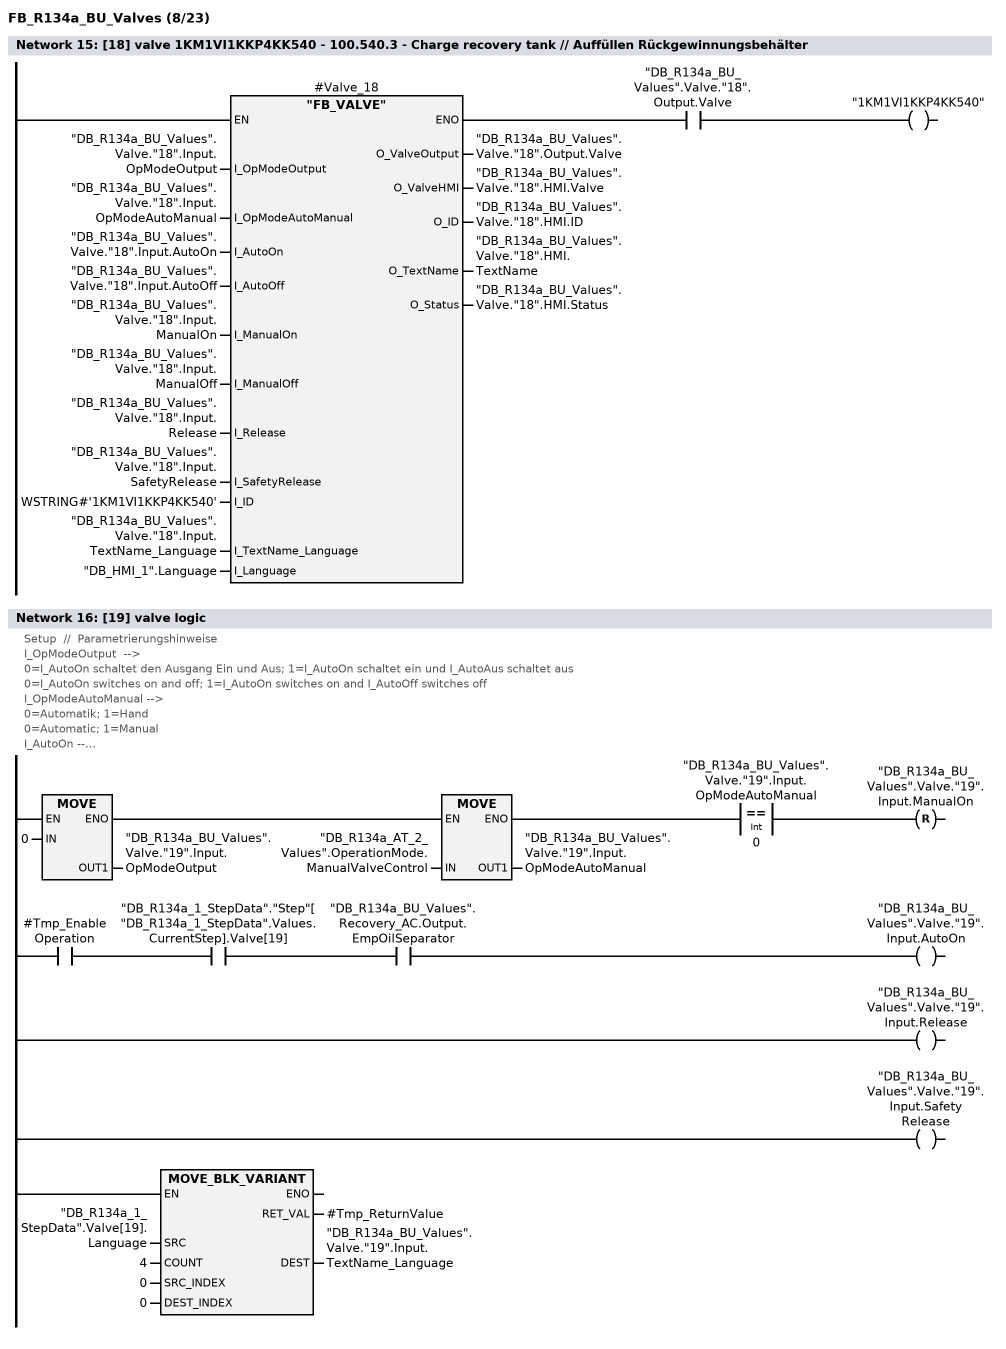
   RUNG wire#powerrail
      #Valve_18(I_OpModeOutput := "DB_R134a_BU_Values".Valve."18".Input.OpModeOutput, I_OpModeAutoManual := "DB_R134a_BU_Values".Valve."18".Input.OpModeAutoManual, I_AutoOn := "DB_R134a_BU_Values".Valve."18".Input.AutoOn, I_AutoOff := "DB_R134a_BU_Values".Valve."18".Input.AutoOff, I_ManualOn := "DB_R134a_BU_Values".Valve."18".Input.ManualOn, I_ManualOff := "DB_R134a_BU_Values".Valve."18".Input.ManualOff, I_Release := "DB_R134a_BU_Values".Valve."18".Input.Release, I_SafetyRelease := "DB_R134a_BU_Values".Valve."18".Input.SafetyRelease, I_ID := WSTRING#'1KM1VI1KKP4KK540', I_TextName_Language := "DB_R134a_BU_Values".Valve."18".Input.TextName_Language, I_Language := "DB_HMI_1".Language, O_ValveOutput => "DB_R134a_BU_Values".Valve."18".Output.Valve, O_ValveHMI => "DB_R134a_BU_Values".Valve."18".HMI.Valve, O_ID => "DB_R134a_BU_Values".Valve."18".HMI.ID, O_TextName => "DB_R134a_BU_Values".Valve."18".HMI.TextName, O_Status => "DB_R134a_BU_Values".Valve."18".HMI.Status)
      Contact( "DB_R134a_BU_Values".Valve."18".Output.Valve )
      Coil( "1KM1VI1KKP4KK540" )
   END_RUNG
   // the same network as SCL:
   #Valve_18(I_OpModeOutput := "DB_R134a_BU_Values".Valve."18".Input.OpModeOutput,   // "FB_VALVE"
             I_OpModeAutoManual := "DB_R134a_BU_Values".Valve."18".Input.OpModeAutoManual,
             I_AutoOn := "DB_R134a_BU_Values".Valve."18".Input.AutoOn,
             I_AutoOff := "DB_R134a_BU_Values".Valve."18".Input.AutoOff,
             I_ManualOn := "DB_R134a_BU_Values".Valve."18".Input.ManualOn,
             I_ManualOff := "DB_R134a_BU_Values".Valve."18".Input.ManualOff,
             I_Release := "DB_R134a_BU_Values".Valve."18".Input.Release,
             I_SafetyRelease := "DB_R134a_BU_Values".Valve."18".Input.SafetyRelease,
             I_ID := WSTRING#'1KM1VI1KKP4KK540',
             I_TextName_Language := "DB_R134a_BU_Values".Valve."18".Input.TextName_Language,
             I_Language := "DB_HMI_1".Language,
             O_ValveOutput => "DB_R134a_BU_Values".Valve."18".Output.Valve,
             O_ValveHMI => "DB_R134a_BU_Values".Valve."18".HMI.Valve,
             O_ID => "DB_R134a_BU_Values".Valve."18".HMI.ID,
             O_TextName => "DB_R134a_BU_Values".Valve."18".HMI.TextName,
             O_Status => "DB_R134a_BU_Values".Valve."18".HMI.Status,
             ENO => #_w1);
   "1KM1VI1KKP4KK540" := #_w1 AND "DB_R134a_BU_Values".Valve."18".Output.Valve;
END_REGION

REGION Network 16: [19] valve logic
   // Setup  //  Parametrierungshinweise
   // I_OpModeOutput  -->
   // 0=I_AutoOn schaltet den Ausgang Ein und Aus; 1=I_AutoOn schaltet ein und I_AutoAus schaltet aus
   // 0=I_AutoOn switches on and off; 1=I_AutoOn switches on and I_AutoOff switches off
   // 
   // I_OpModeAutoManual -->
   // 0=Automatik; 1=Hand
   // 0=Automatic; 1=Manual
   // 
   // I_AutoOn -->
   // 1=Automatik Ein, Eingang für die normalen Ventilverschaltungsbedingungen
   // 1=Automatic On, Input for the normal valve conditions
   // 
   // I_Release -->
   // 1=Freigabe, Eingang für die Fehlerbedingungen
   // 1=Release, Input for fault conditions
   // 
   // I_SafetyRelease -->
   // 1=Sicherheitsfreigabe, Eingang für zusätzliche Schaltbefehle aus dem Sicherheitsprogramm
   // 1=Safety release, Input for additional safety conditions from the safety program
   RUNG wire#powerrail
      Move(in := 0, out1 => "DB_R134a_BU_Values".Valve."19".Input.OpModeOutput)
      Move(in := "DB_R134a_AT_2_Values".OperationMode.ManualValveControl, out1 => "DB_R134a_BU_Values".Valve."19".Input.OpModeAutoManual)
      { S7_Templates := "SrcType := Int" } EQ_Contact(in1 := "DB_R134a_BU_Values".Valve."19".Input.OpModeAutoManual, in2 := 0)
      R_Coil( "DB_R134a_BU_Values".Valve."19".Input.ManualOn )
   END_RUNG
   RUNG wire#powerrail
      Contact( #Tmp_EnableOperation )
      Contact( "DB_R134a_1_StepData"."Step"["DB_R134a_1_StepData".Values.CurrentStep].Valve[19] )
      Contact( "DB_R134a_BU_Values".Recovery_AC.Output.EmpOilSeparator )
      Coil( "DB_R134a_BU_Values".Valve."19".Input.AutoOn )
   END_RUNG
   RUNG wire#powerrail
      Coil( "DB_R134a_BU_Values".Valve."19".Input.Release )
   END_RUNG
   RUNG wire#powerrail
      Coil( "DB_R134a_BU_Values".Valve."19".Input.SafetyRelease )
   END_RUNG
   RUNG wire#powerrail
      MOVE_BLK_VARIANT(SRC := "DB_R134a_1_StepData".Valve[19].Language, COUNT := 4, SRC_INDEX := 0, DEST_INDEX := 0, Ret_Val => #Tmp_ReturnValue, DEST => "DB_R134a_BU_Values".Valve."19".Input.TextName_Language)
   END_RUNG
   // the same network as SCL:
   "DB_R134a_BU_Values".Valve."19".Input.OpModeOutput := 0;
   "DB_R134a_BU_Values".Valve."19".Input.OpModeAutoManual := "DB_R134a_AT_2_Values".OperationMode.ManualValveControl;
   IF "DB_R134a_BU_Values".Valve."19".Input.OpModeAutoManual = 0 THEN
       "DB_R134a_BU_Values".Valve."19".Input.ManualOn := FALSE;
   END_IF;
   "DB_R134a_BU_Values".Valve."19".Input.AutoOn := #Tmp_EnableOperation AND "DB_R134a_1_StepData"."Step"["DB_R134a_1_StepData".Values.CurrentStep].Valve[19] AND "DB_R134a_BU_Values".Recovery_AC.Output.EmpOilSeparator;
   "DB_R134a_BU_Values".Valve."19".Input.Release := TRUE;
   "DB_R134a_BU_Values".Valve."19".Input.SafetyRelease := TRUE;
   #Tmp_ReturnValue := MOVE_BLK_VARIANT(SRC := "DB_R134a_1_StepData".Valve[19].Language,
                           COUNT := 4,
                           SRC_INDEX := 0,
                           DEST_INDEX := 0,
                           DEST => "DB_R134a_BU_Values".Valve."19".Input.TextName_Language);
END_REGION

REGION Network 17: [19] valve 1KM1VI1KKP6KK520 - 108.520.3 - Discharge separator // Entleeren Abscheidebehälter
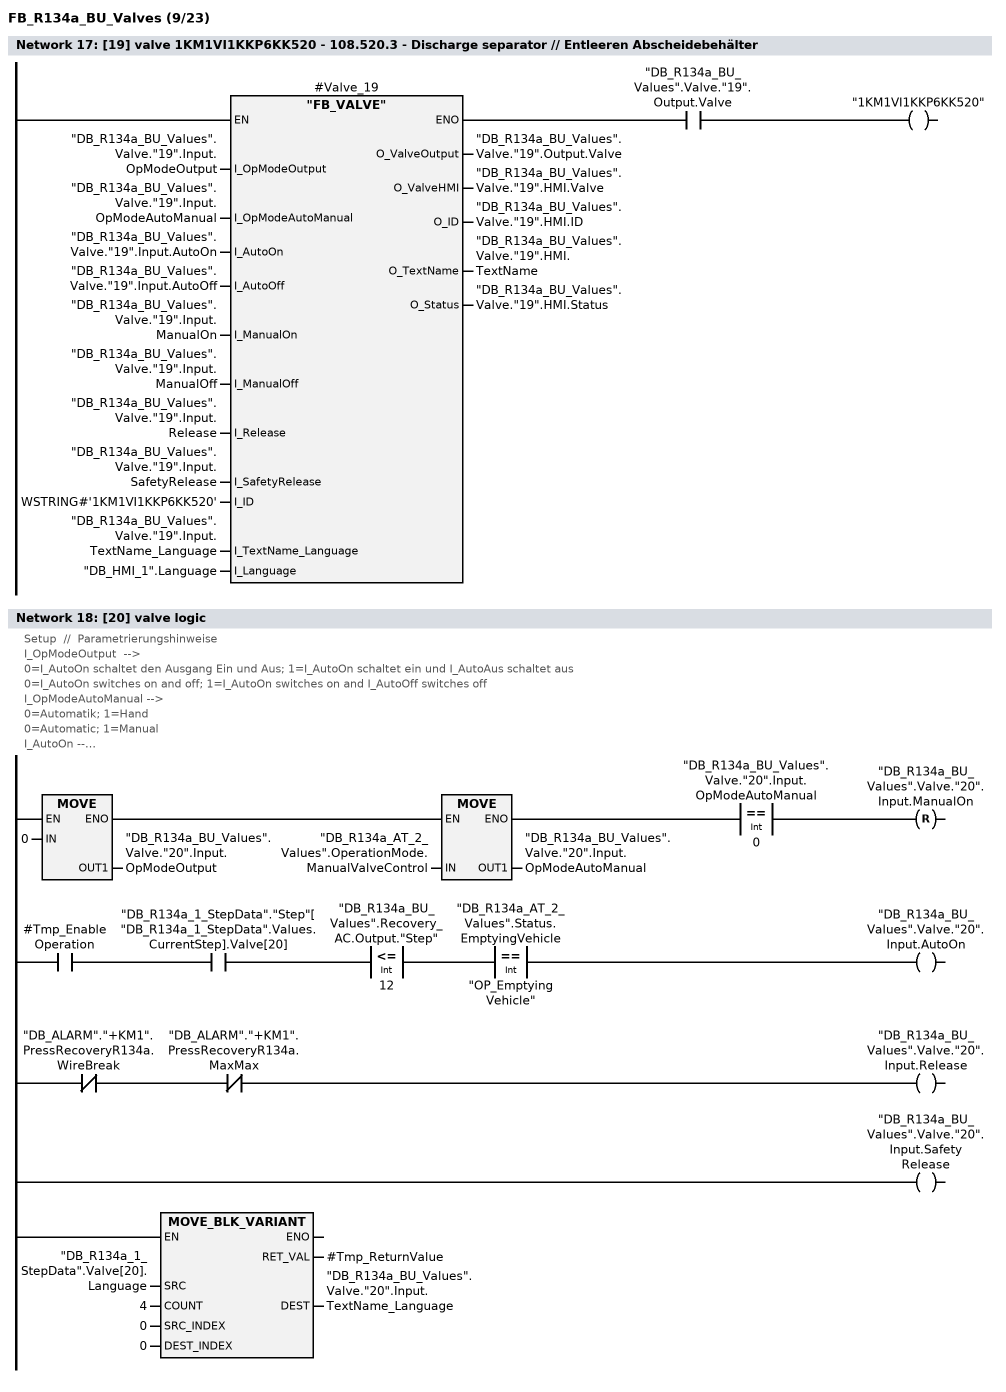
   RUNG wire#powerrail
      #Valve_19(I_OpModeOutput := "DB_R134a_BU_Values".Valve."19".Input.OpModeOutput, I_OpModeAutoManual := "DB_R134a_BU_Values".Valve."19".Input.OpModeAutoManual, I_AutoOn := "DB_R134a_BU_Values".Valve."19".Input.AutoOn, I_AutoOff := "DB_R134a_BU_Values".Valve."19".Input.AutoOff, I_ManualOn := "DB_R134a_BU_Values".Valve."19".Input.ManualOn, I_ManualOff := "DB_R134a_BU_Values".Valve."19".Input.ManualOff, I_Release := "DB_R134a_BU_Values".Valve."19".Input.Release, I_SafetyRelease := "DB_R134a_BU_Values".Valve."19".Input.SafetyRelease, I_ID := WSTRING#'1KM1VI1KKP6KK520', I_TextName_Language := "DB_R134a_BU_Values".Valve."19".Input.TextName_Language, I_Language := "DB_HMI_1".Language, O_ValveOutput => "DB_R134a_BU_Values".Valve."19".Output.Valve, O_ValveHMI => "DB_R134a_BU_Values".Valve."19".HMI.Valve, O_ID => "DB_R134a_BU_Values".Valve."19".HMI.ID, O_TextName => "DB_R134a_BU_Values".Valve."19".HMI.TextName, O_Status => "DB_R134a_BU_Values".Valve."19".HMI.Status)
      Contact( "DB_R134a_BU_Values".Valve."19".Output.Valve )
      Coil( "1KM1VI1KKP6KK520" )
   END_RUNG
   // the same network as SCL:
   #Valve_19(I_OpModeOutput := "DB_R134a_BU_Values".Valve."19".Input.OpModeOutput,   // "FB_VALVE"
             I_OpModeAutoManual := "DB_R134a_BU_Values".Valve."19".Input.OpModeAutoManual,
             I_AutoOn := "DB_R134a_BU_Values".Valve."19".Input.AutoOn,
             I_AutoOff := "DB_R134a_BU_Values".Valve."19".Input.AutoOff,
             I_ManualOn := "DB_R134a_BU_Values".Valve."19".Input.ManualOn,
             I_ManualOff := "DB_R134a_BU_Values".Valve."19".Input.ManualOff,
             I_Release := "DB_R134a_BU_Values".Valve."19".Input.Release,
             I_SafetyRelease := "DB_R134a_BU_Values".Valve."19".Input.SafetyRelease,
             I_ID := WSTRING#'1KM1VI1KKP6KK520',
             I_TextName_Language := "DB_R134a_BU_Values".Valve."19".Input.TextName_Language,
             I_Language := "DB_HMI_1".Language,
             O_ValveOutput => "DB_R134a_BU_Values".Valve."19".Output.Valve,
             O_ValveHMI => "DB_R134a_BU_Values".Valve."19".HMI.Valve,
             O_ID => "DB_R134a_BU_Values".Valve."19".HMI.ID,
             O_TextName => "DB_R134a_BU_Values".Valve."19".HMI.TextName,
             O_Status => "DB_R134a_BU_Values".Valve."19".HMI.Status,
             ENO => #_w1);
   "1KM1VI1KKP6KK520" := #_w1 AND "DB_R134a_BU_Values".Valve."19".Output.Valve;
END_REGION

REGION Network 18: [20] valve logic
   // Setup  //  Parametrierungshinweise
   // I_OpModeOutput  -->
   // 0=I_AutoOn schaltet den Ausgang Ein und Aus; 1=I_AutoOn schaltet ein und I_AutoAus schaltet aus
   // 0=I_AutoOn switches on and off; 1=I_AutoOn switches on and I_AutoOff switches off
   // 
   // I_OpModeAutoManual -->
   // 0=Automatik; 1=Hand
   // 0=Automatic; 1=Manual
   // 
   // I_AutoOn -->
   // 1=Automatik Ein, Eingang für die normalen Ventilverschaltungsbedingungen
   // 1=Automatic On, Input for the normal valve conditions
   // 
   // I_Release -->
   // 1=Freigabe, Eingang für die Fehlerbedingungen
   // 1=Release, Input for fault conditions
   // 
   // I_SafetyRelease -->
   // 1=Sicherheitsfreigabe, Eingang für zusätzliche Schaltbefehle aus dem Sicherheitsprogramm
   // 1=Safety release, Input for additional safety conditions from the safety program
   RUNG wire#powerrail
      Move(in := 0, out1 => "DB_R134a_BU_Values".Valve."20".Input.OpModeOutput)
      Move(in := "DB_R134a_AT_2_Values".OperationMode.ManualValveControl, out1 => "DB_R134a_BU_Values".Valve."20".Input.OpModeAutoManual)
      { S7_Templates := "SrcType := Int" } EQ_Contact(in1 := "DB_R134a_BU_Values".Valve."20".Input.OpModeAutoManual, in2 := 0)
      R_Coil( "DB_R134a_BU_Values".Valve."20".Input.ManualOn )
   END_RUNG
   RUNG wire#powerrail
      Contact( #Tmp_EnableOperation )
      Contact( "DB_R134a_1_StepData"."Step"["DB_R134a_1_StepData".Values.CurrentStep].Valve[20] )
      { S7_Templates := "SrcType := Int" } LE_Contact(in1 := "DB_R134a_BU_Values".Recovery_AC.Output."Step", in2 := 12)
      { S7_Templates := "SrcType := Int" } EQ_Contact(in1 := "DB_R134a_AT_2_Values".Status.EmptyingVehicle, in2 := "OP_EmptyingVehicle")
      Coil( "DB_R134a_BU_Values".Valve."20".Input.AutoOn )
   END_RUNG
   RUNG wire#powerrail
      I_Contact( "DB_ALARM"."+KM1".PressRecoveryR134a.WireBreak )
      I_Contact( "DB_ALARM"."+KM1".PressRecoveryR134a.MaxMax )
      Coil( "DB_R134a_BU_Values".Valve."20".Input.Release )
   END_RUNG
   RUNG wire#powerrail
      Coil( "DB_R134a_BU_Values".Valve."20".Input.SafetyRelease )
   END_RUNG
   RUNG wire#powerrail
      MOVE_BLK_VARIANT(SRC := "DB_R134a_1_StepData".Valve[20].Language, COUNT := 4, SRC_INDEX := 0, DEST_INDEX := 0, Ret_Val => #Tmp_ReturnValue, DEST => "DB_R134a_BU_Values".Valve."20".Input.TextName_Language)
   END_RUNG
   // the same network as SCL:
   "DB_R134a_BU_Values".Valve."20".Input.OpModeOutput := 0;
   "DB_R134a_BU_Values".Valve."20".Input.OpModeAutoManual := "DB_R134a_AT_2_Values".OperationMode.ManualValveControl;
   IF "DB_R134a_BU_Values".Valve."20".Input.OpModeAutoManual = 0 THEN
       "DB_R134a_BU_Values".Valve."20".Input.ManualOn := FALSE;
   END_IF;
   "DB_R134a_BU_Values".Valve."20".Input.AutoOn := #Tmp_EnableOperation AND "DB_R134a_1_StepData"."Step"["DB_R134a_1_StepData".Values.CurrentStep].Valve[20] AND ("DB_R134a_BU_Values".Recovery_AC.Output."Step" <= 12) AND ("DB_R134a_AT_2_Values".Status.EmptyingVehicle = "OP_EmptyingVehicle");
   "DB_R134a_BU_Values".Valve."20".Input.Release := NOT "DB_ALARM"."+KM1".PressRecoveryR134a.WireBreak AND NOT "DB_ALARM"."+KM1".PressRecoveryR134a.MaxMax;
   "DB_R134a_BU_Values".Valve."20".Input.SafetyRelease := TRUE;
   #Tmp_ReturnValue := MOVE_BLK_VARIANT(SRC := "DB_R134a_1_StepData".Valve[20].Language,
                           COUNT := 4,
                           SRC_INDEX := 0,
                           DEST_INDEX := 0,
                           DEST => "DB_R134a_BU_Values".Valve."20".Input.TextName_Language);
END_REGION

REGION Network 19: [20] valve 1KM1VI1KKP4KK380 - 108.380.3 - Recovery - near system // Rückgewinnung / Rückgewinnung 1 - nahe System
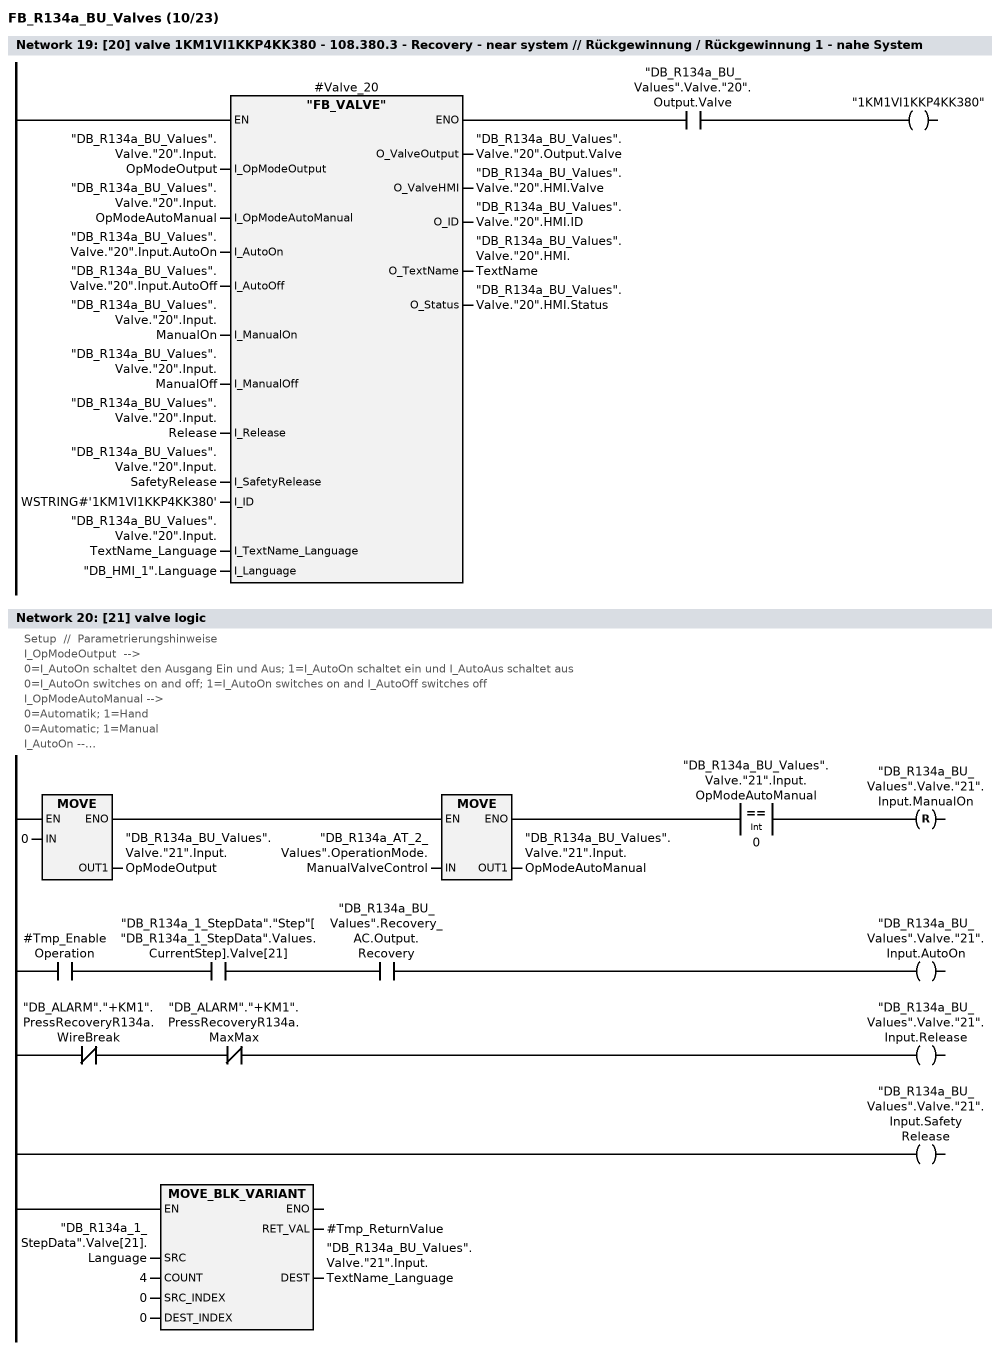
   RUNG wire#powerrail
      #Valve_20(I_OpModeOutput := "DB_R134a_BU_Values".Valve."20".Input.OpModeOutput, I_OpModeAutoManual := "DB_R134a_BU_Values".Valve."20".Input.OpModeAutoManual, I_AutoOn := "DB_R134a_BU_Values".Valve."20".Input.AutoOn, I_AutoOff := "DB_R134a_BU_Values".Valve."20".Input.AutoOff, I_ManualOn := "DB_R134a_BU_Values".Valve."20".Input.ManualOn, I_ManualOff := "DB_R134a_BU_Values".Valve."20".Input.ManualOff, I_Release := "DB_R134a_BU_Values".Valve."20".Input.Release, I_SafetyRelease := "DB_R134a_BU_Values".Valve."20".Input.SafetyRelease, I_ID := WSTRING#'1KM1VI1KKP4KK380', I_TextName_Language := "DB_R134a_BU_Values".Valve."20".Input.TextName_Language, I_Language := "DB_HMI_1".Language, O_ValveOutput => "DB_R134a_BU_Values".Valve."20".Output.Valve, O_ValveHMI => "DB_R134a_BU_Values".Valve."20".HMI.Valve, O_ID => "DB_R134a_BU_Values".Valve."20".HMI.ID, O_TextName => "DB_R134a_BU_Values".Valve."20".HMI.TextName, O_Status => "DB_R134a_BU_Values".Valve."20".HMI.Status)
      Contact( "DB_R134a_BU_Values".Valve."20".Output.Valve )
      Coil( "1KM1VI1KKP4KK380" )
   END_RUNG
   // the same network as SCL:
   #Valve_20(I_OpModeOutput := "DB_R134a_BU_Values".Valve."20".Input.OpModeOutput,   // "FB_VALVE"
             I_OpModeAutoManual := "DB_R134a_BU_Values".Valve."20".Input.OpModeAutoManual,
             I_AutoOn := "DB_R134a_BU_Values".Valve."20".Input.AutoOn,
             I_AutoOff := "DB_R134a_BU_Values".Valve."20".Input.AutoOff,
             I_ManualOn := "DB_R134a_BU_Values".Valve."20".Input.ManualOn,
             I_ManualOff := "DB_R134a_BU_Values".Valve."20".Input.ManualOff,
             I_Release := "DB_R134a_BU_Values".Valve."20".Input.Release,
             I_SafetyRelease := "DB_R134a_BU_Values".Valve."20".Input.SafetyRelease,
             I_ID := WSTRING#'1KM1VI1KKP4KK380',
             I_TextName_Language := "DB_R134a_BU_Values".Valve."20".Input.TextName_Language,
             I_Language := "DB_HMI_1".Language,
             O_ValveOutput => "DB_R134a_BU_Values".Valve."20".Output.Valve,
             O_ValveHMI => "DB_R134a_BU_Values".Valve."20".HMI.Valve,
             O_ID => "DB_R134a_BU_Values".Valve."20".HMI.ID,
             O_TextName => "DB_R134a_BU_Values".Valve."20".HMI.TextName,
             O_Status => "DB_R134a_BU_Values".Valve."20".HMI.Status,
             ENO => #_w1);
   "1KM1VI1KKP4KK380" := #_w1 AND "DB_R134a_BU_Values".Valve."20".Output.Valve;
END_REGION

REGION Network 20: [21] valve logic
   // Setup  //  Parametrierungshinweise
   // I_OpModeOutput  -->
   // 0=I_AutoOn schaltet den Ausgang Ein und Aus; 1=I_AutoOn schaltet ein und I_AutoAus schaltet aus
   // 0=I_AutoOn switches on and off; 1=I_AutoOn switches on and I_AutoOff switches off
   // 
   // I_OpModeAutoManual -->
   // 0=Automatik; 1=Hand
   // 0=Automatic; 1=Manual
   // 
   // I_AutoOn -->
   // 1=Automatik Ein, Eingang für die normalen Ventilverschaltungsbedingungen
   // 1=Automatic On, Input for the normal valve conditions
   // 
   // I_Release -->
   // 1=Freigabe, Eingang für die Fehlerbedingungen
   // 1=Release, Input for fault conditions
   // 
   // I_SafetyRelease -->
   // 1=Sicherheitsfreigabe, Eingang für zusätzliche Schaltbefehle aus dem Sicherheitsprogramm
   // 1=Safety release, Input for additional safety conditions from the safety program
   RUNG wire#powerrail
      Move(in := 0, out1 => "DB_R134a_BU_Values".Valve."21".Input.OpModeOutput)
      Move(in := "DB_R134a_AT_2_Values".OperationMode.ManualValveControl, out1 => "DB_R134a_BU_Values".Valve."21".Input.OpModeAutoManual)
      { S7_Templates := "SrcType := Int" } EQ_Contact(in1 := "DB_R134a_BU_Values".Valve."21".Input.OpModeAutoManual, in2 := 0)
      R_Coil( "DB_R134a_BU_Values".Valve."21".Input.ManualOn )
   END_RUNG
   RUNG wire#powerrail
      Contact( #Tmp_EnableOperation )
      Contact( "DB_R134a_1_StepData"."Step"["DB_R134a_1_StepData".Values.CurrentStep].Valve[21] )
      Contact( "DB_R134a_BU_Values".Recovery_AC.Output.Recovery )
      Coil( "DB_R134a_BU_Values".Valve."21".Input.AutoOn )
   END_RUNG
   RUNG wire#powerrail
      I_Contact( "DB_ALARM"."+KM1".PressRecoveryR134a.WireBreak )
      I_Contact( "DB_ALARM"."+KM1".PressRecoveryR134a.MaxMax )
      Coil( "DB_R134a_BU_Values".Valve."21".Input.Release )
   END_RUNG
   RUNG wire#powerrail
      Coil( "DB_R134a_BU_Values".Valve."21".Input.SafetyRelease )
   END_RUNG
   RUNG wire#powerrail
      MOVE_BLK_VARIANT(SRC := "DB_R134a_1_StepData".Valve[21].Language, COUNT := 4, SRC_INDEX := 0, DEST_INDEX := 0, Ret_Val => #Tmp_ReturnValue, DEST => "DB_R134a_BU_Values".Valve."21".Input.TextName_Language)
   END_RUNG
   // the same network as SCL:
   "DB_R134a_BU_Values".Valve."21".Input.OpModeOutput := 0;
   "DB_R134a_BU_Values".Valve."21".Input.OpModeAutoManual := "DB_R134a_AT_2_Values".OperationMode.ManualValveControl;
   IF "DB_R134a_BU_Values".Valve."21".Input.OpModeAutoManual = 0 THEN
       "DB_R134a_BU_Values".Valve."21".Input.ManualOn := FALSE;
   END_IF;
   "DB_R134a_BU_Values".Valve."21".Input.AutoOn := #Tmp_EnableOperation AND "DB_R134a_1_StepData"."Step"["DB_R134a_1_StepData".Values.CurrentStep].Valve[21] AND "DB_R134a_BU_Values".Recovery_AC.Output.Recovery;
   "DB_R134a_BU_Values".Valve."21".Input.Release := NOT "DB_ALARM"."+KM1".PressRecoveryR134a.WireBreak AND NOT "DB_ALARM"."+KM1".PressRecoveryR134a.MaxMax;
   "DB_R134a_BU_Values".Valve."21".Input.SafetyRelease := TRUE;
   #Tmp_ReturnValue := MOVE_BLK_VARIANT(SRC := "DB_R134a_1_StepData".Valve[21].Language,
                           COUNT := 4,
                           SRC_INDEX := 0,
                           DEST_INDEX := 0,
                           DEST => "DB_R134a_BU_Values".Valve."21".Input.TextName_Language);
END_REGION

REGION Network 21: [21] valve 1KM1VI1KKP6KK381 - 100.381.3 - Recovery - near tank // Rückgewinnung 2 - nahe Speicher
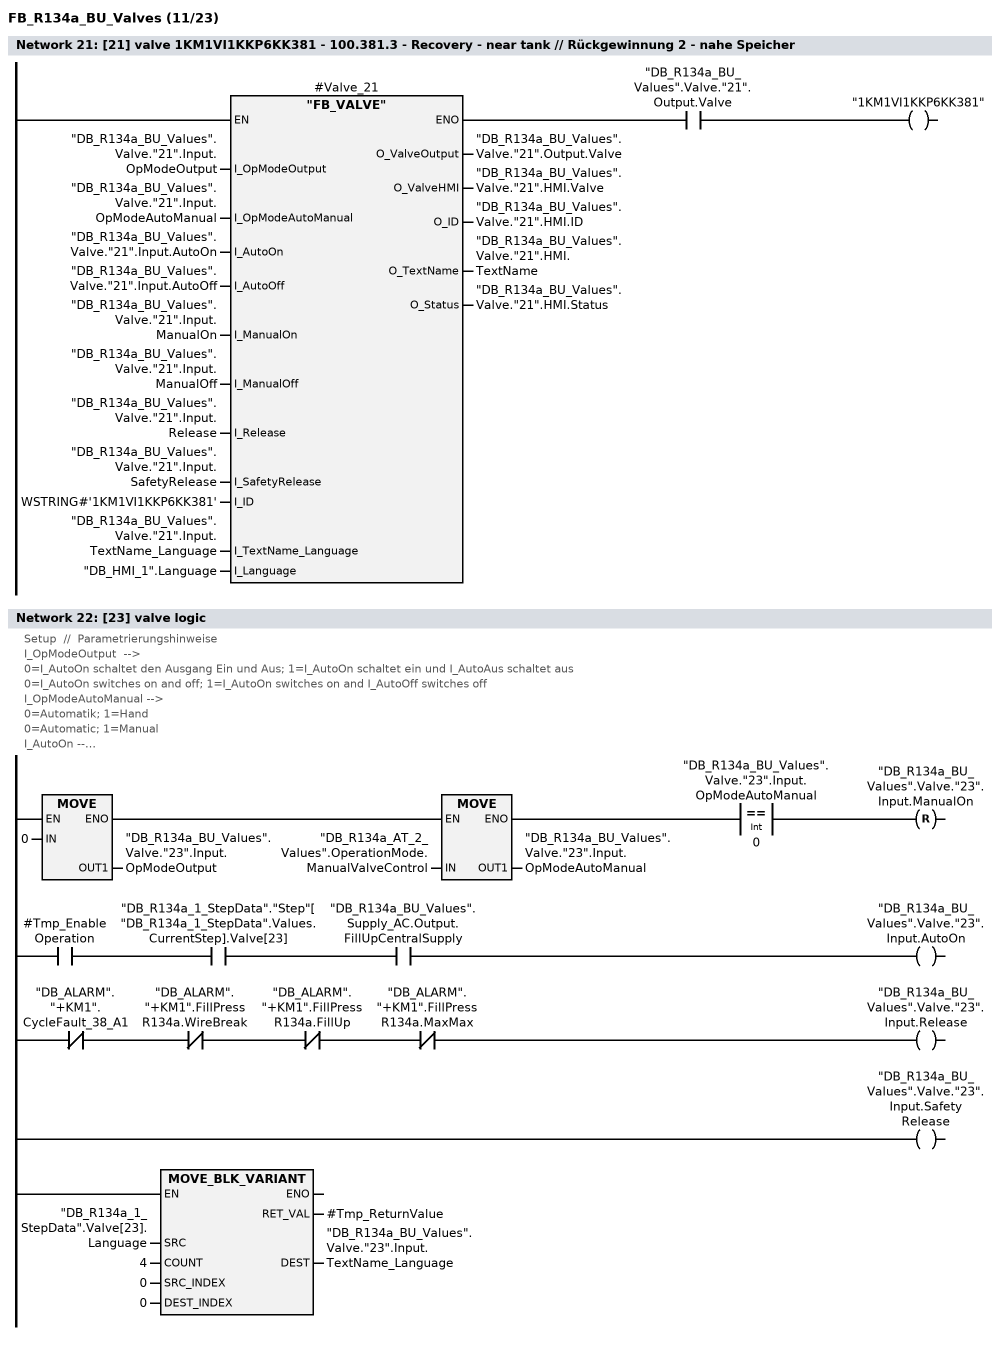
   RUNG wire#powerrail
      #Valve_21(I_OpModeOutput := "DB_R134a_BU_Values".Valve."21".Input.OpModeOutput, I_OpModeAutoManual := "DB_R134a_BU_Values".Valve."21".Input.OpModeAutoManual, I_AutoOn := "DB_R134a_BU_Values".Valve."21".Input.AutoOn, I_AutoOff := "DB_R134a_BU_Values".Valve."21".Input.AutoOff, I_ManualOn := "DB_R134a_BU_Values".Valve."21".Input.ManualOn, I_ManualOff := "DB_R134a_BU_Values".Valve."21".Input.ManualOff, I_Release := "DB_R134a_BU_Values".Valve."21".Input.Release, I_SafetyRelease := "DB_R134a_BU_Values".Valve."21".Input.SafetyRelease, I_ID := WSTRING#'1KM1VI1KKP6KK381', I_TextName_Language := "DB_R134a_BU_Values".Valve."21".Input.TextName_Language, I_Language := "DB_HMI_1".Language, O_ValveOutput => "DB_R134a_BU_Values".Valve."21".Output.Valve, O_ValveHMI => "DB_R134a_BU_Values".Valve."21".HMI.Valve, O_ID => "DB_R134a_BU_Values".Valve."21".HMI.ID, O_TextName => "DB_R134a_BU_Values".Valve."21".HMI.TextName, O_Status => "DB_R134a_BU_Values".Valve."21".HMI.Status)
      Contact( "DB_R134a_BU_Values".Valve."21".Output.Valve )
      Coil( "1KM1VI1KKP6KK381" )
   END_RUNG
   // the same network as SCL:
   #Valve_21(I_OpModeOutput := "DB_R134a_BU_Values".Valve."21".Input.OpModeOutput,   // "FB_VALVE"
             I_OpModeAutoManual := "DB_R134a_BU_Values".Valve."21".Input.OpModeAutoManual,
             I_AutoOn := "DB_R134a_BU_Values".Valve."21".Input.AutoOn,
             I_AutoOff := "DB_R134a_BU_Values".Valve."21".Input.AutoOff,
             I_ManualOn := "DB_R134a_BU_Values".Valve."21".Input.ManualOn,
             I_ManualOff := "DB_R134a_BU_Values".Valve."21".Input.ManualOff,
             I_Release := "DB_R134a_BU_Values".Valve."21".Input.Release,
             I_SafetyRelease := "DB_R134a_BU_Values".Valve."21".Input.SafetyRelease,
             I_ID := WSTRING#'1KM1VI1KKP6KK381',
             I_TextName_Language := "DB_R134a_BU_Values".Valve."21".Input.TextName_Language,
             I_Language := "DB_HMI_1".Language,
             O_ValveOutput => "DB_R134a_BU_Values".Valve."21".Output.Valve,
             O_ValveHMI => "DB_R134a_BU_Values".Valve."21".HMI.Valve,
             O_ID => "DB_R134a_BU_Values".Valve."21".HMI.ID,
             O_TextName => "DB_R134a_BU_Values".Valve."21".HMI.TextName,
             O_Status => "DB_R134a_BU_Values".Valve."21".HMI.Status,
             ENO => #_w1);
   "1KM1VI1KKP6KK381" := #_w1 AND "DB_R134a_BU_Values".Valve."21".Output.Valve;
END_REGION

REGION Network 22: [23] valve logic
   // Setup  //  Parametrierungshinweise
   // I_OpModeOutput  -->
   // 0=I_AutoOn schaltet den Ausgang Ein und Aus; 1=I_AutoOn schaltet ein und I_AutoAus schaltet aus
   // 0=I_AutoOn switches on and off; 1=I_AutoOn switches on and I_AutoOff switches off
   // 
   // I_OpModeAutoManual -->
   // 0=Automatik; 1=Hand
   // 0=Automatic; 1=Manual
   // 
   // I_AutoOn -->
   // 1=Automatik Ein, Eingang für die normalen Ventilverschaltungsbedingungen
   // 1=Automatic On, Input for the normal valve conditions
   // 
   // I_Release -->
   // 1=Freigabe, Eingang für die Fehlerbedingungen
   // 1=Release, Input for fault conditions
   // 
   // I_SafetyRelease -->
   // 1=Sicherheitsfreigabe, Eingang für zusätzliche Schaltbefehle aus dem Sicherheitsprogramm
   // 1=Safety release, Input for additional safety conditions from the safety program
   RUNG wire#powerrail
      Move(in := 0, out1 => "DB_R134a_BU_Values".Valve."23".Input.OpModeOutput)
      Move(in := "DB_R134a_AT_2_Values".OperationMode.ManualValveControl, out1 => "DB_R134a_BU_Values".Valve."23".Input.OpModeAutoManual)
      { S7_Templates := "SrcType := Int" } EQ_Contact(in1 := "DB_R134a_BU_Values".Valve."23".Input.OpModeAutoManual, in2 := 0)
      R_Coil( "DB_R134a_BU_Values".Valve."23".Input.ManualOn )
   END_RUNG
   RUNG wire#powerrail
      Contact( #Tmp_EnableOperation )
      Contact( "DB_R134a_1_StepData"."Step"["DB_R134a_1_StepData".Values.CurrentStep].Valve[23] )
      Contact( "DB_R134a_BU_Values".Supply_AC.Output.FillUpCentralSupply )
      Coil( "DB_R134a_BU_Values".Valve."23".Input.AutoOn )
   END_RUNG
   RUNG wire#powerrail
      I_Contact( "DB_ALARM"."+KM1".CycleFault_38_A1 )
      I_Contact( "DB_ALARM"."+KM1".FillPressR134a.WireBreak )
      I_Contact( "DB_ALARM"."+KM1".FillPressR134a.FillUp )
      I_Contact( "DB_ALARM"."+KM1".FillPressR134a.MaxMax )
      Coil( "DB_R134a_BU_Values".Valve."23".Input.Release )
   END_RUNG
   RUNG wire#powerrail
      Coil( "DB_R134a_BU_Values".Valve."23".Input.SafetyRelease )
   END_RUNG
   RUNG wire#powerrail
      MOVE_BLK_VARIANT(SRC := "DB_R134a_1_StepData".Valve[23].Language, COUNT := 4, SRC_INDEX := 0, DEST_INDEX := 0, Ret_Val => #Tmp_ReturnValue, DEST => "DB_R134a_BU_Values".Valve."23".Input.TextName_Language)
   END_RUNG
   // the same network as SCL:
   "DB_R134a_BU_Values".Valve."23".Input.OpModeOutput := 0;
   "DB_R134a_BU_Values".Valve."23".Input.OpModeAutoManual := "DB_R134a_AT_2_Values".OperationMode.ManualValveControl;
   IF "DB_R134a_BU_Values".Valve."23".Input.OpModeAutoManual = 0 THEN
       "DB_R134a_BU_Values".Valve."23".Input.ManualOn := FALSE;
   END_IF;
   "DB_R134a_BU_Values".Valve."23".Input.AutoOn := #Tmp_EnableOperation AND "DB_R134a_1_StepData"."Step"["DB_R134a_1_StepData".Values.CurrentStep].Valve[23] AND "DB_R134a_BU_Values".Supply_AC.Output.FillUpCentralSupply;
   "DB_R134a_BU_Values".Valve."23".Input.Release := NOT "DB_ALARM"."+KM1".CycleFault_38_A1 AND NOT "DB_ALARM"."+KM1".FillPressR134a.WireBreak AND NOT "DB_ALARM"."+KM1".FillPressR134a.FillUp AND NOT "DB_ALARM"."+KM1".FillPressR134a.MaxMax;
   "DB_R134a_BU_Values".Valve."23".Input.SafetyRelease := TRUE;
   #Tmp_ReturnValue := MOVE_BLK_VARIANT(SRC := "DB_R134a_1_StepData".Valve[23].Language,
                           COUNT := 4,
                           SRC_INDEX := 0,
                           DEST_INDEX := 0,
                           DEST => "DB_R134a_BU_Values".Valve."23".Input.TextName_Language);
END_REGION

REGION Network 23: [23] valve 1KM1VI1KKP2KK20 - 100.20.3 - Supply central // Versorgung - zentral
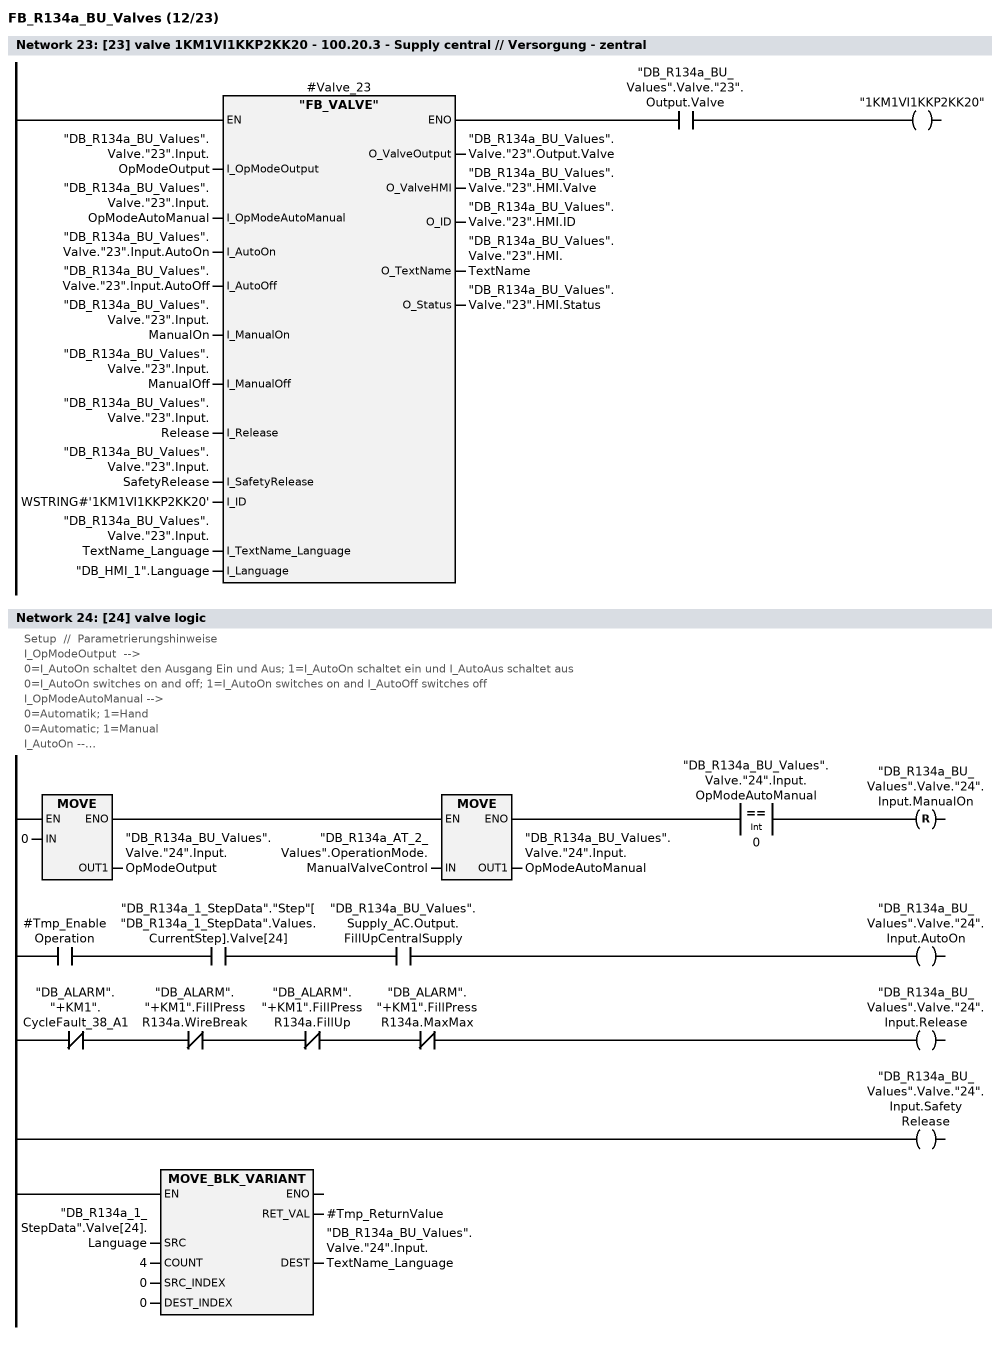
   RUNG wire#powerrail
      #Valve_23(I_OpModeOutput := "DB_R134a_BU_Values".Valve."23".Input.OpModeOutput, I_OpModeAutoManual := "DB_R134a_BU_Values".Valve."23".Input.OpModeAutoManual, I_AutoOn := "DB_R134a_BU_Values".Valve."23".Input.AutoOn, I_AutoOff := "DB_R134a_BU_Values".Valve."23".Input.AutoOff, I_ManualOn := "DB_R134a_BU_Values".Valve."23".Input.ManualOn, I_ManualOff := "DB_R134a_BU_Values".Valve."23".Input.ManualOff, I_Release := "DB_R134a_BU_Values".Valve."23".Input.Release, I_SafetyRelease := "DB_R134a_BU_Values".Valve."23".Input.SafetyRelease, I_ID := WSTRING#'1KM1VI1KKP2KK20', I_TextName_Language := "DB_R134a_BU_Values".Valve."23".Input.TextName_Language, I_Language := "DB_HMI_1".Language, O_ValveOutput => "DB_R134a_BU_Values".Valve."23".Output.Valve, O_ValveHMI => "DB_R134a_BU_Values".Valve."23".HMI.Valve, O_ID => "DB_R134a_BU_Values".Valve."23".HMI.ID, O_TextName => "DB_R134a_BU_Values".Valve."23".HMI.TextName, O_Status => "DB_R134a_BU_Values".Valve."23".HMI.Status)
      Contact( "DB_R134a_BU_Values".Valve."23".Output.Valve )
      Coil( "1KM1VI1KKP2KK20" )
   END_RUNG
   // the same network as SCL:
   #Valve_23(I_OpModeOutput := "DB_R134a_BU_Values".Valve."23".Input.OpModeOutput,   // "FB_VALVE"
             I_OpModeAutoManual := "DB_R134a_BU_Values".Valve."23".Input.OpModeAutoManual,
             I_AutoOn := "DB_R134a_BU_Values".Valve."23".Input.AutoOn,
             I_AutoOff := "DB_R134a_BU_Values".Valve."23".Input.AutoOff,
             I_ManualOn := "DB_R134a_BU_Values".Valve."23".Input.ManualOn,
             I_ManualOff := "DB_R134a_BU_Values".Valve."23".Input.ManualOff,
             I_Release := "DB_R134a_BU_Values".Valve."23".Input.Release,
             I_SafetyRelease := "DB_R134a_BU_Values".Valve."23".Input.SafetyRelease,
             I_ID := WSTRING#'1KM1VI1KKP2KK20',
             I_TextName_Language := "DB_R134a_BU_Values".Valve."23".Input.TextName_Language,
             I_Language := "DB_HMI_1".Language,
             O_ValveOutput => "DB_R134a_BU_Values".Valve."23".Output.Valve,
             O_ValveHMI => "DB_R134a_BU_Values".Valve."23".HMI.Valve,
             O_ID => "DB_R134a_BU_Values".Valve."23".HMI.ID,
             O_TextName => "DB_R134a_BU_Values".Valve."23".HMI.TextName,
             O_Status => "DB_R134a_BU_Values".Valve."23".HMI.Status,
             ENO => #_w1);
   "1KM1VI1KKP2KK20" := #_w1 AND "DB_R134a_BU_Values".Valve."23".Output.Valve;
END_REGION

REGION Network 24: [24] valve logic
   // Setup  //  Parametrierungshinweise
   // I_OpModeOutput  -->
   // 0=I_AutoOn schaltet den Ausgang Ein und Aus; 1=I_AutoOn schaltet ein und I_AutoAus schaltet aus
   // 0=I_AutoOn switches on and off; 1=I_AutoOn switches on and I_AutoOff switches off
   // 
   // I_OpModeAutoManual -->
   // 0=Automatik; 1=Hand
   // 0=Automatic; 1=Manual
   // 
   // I_AutoOn -->
   // 1=Automatik Ein, Eingang für die normalen Ventilverschaltungsbedingungen
   // 1=Automatic On, Input for the normal valve conditions
   // 
   // I_Release -->
   // 1=Freigabe, Eingang für die Fehlerbedingungen
   // 1=Release, Input for fault conditions
   // 
   // I_SafetyRelease -->
   // 1=Sicherheitsfreigabe, Eingang für zusätzliche Schaltbefehle aus dem Sicherheitsprogramm
   // 1=Safety release, Input for additional safety conditions from the safety program
   RUNG wire#powerrail
      Move(in := 0, out1 => "DB_R134a_BU_Values".Valve."24".Input.OpModeOutput)
      Move(in := "DB_R134a_AT_2_Values".OperationMode.ManualValveControl, out1 => "DB_R134a_BU_Values".Valve."24".Input.OpModeAutoManual)
      { S7_Templates := "SrcType := Int" } EQ_Contact(in1 := "DB_R134a_BU_Values".Valve."24".Input.OpModeAutoManual, in2 := 0)
      R_Coil( "DB_R134a_BU_Values".Valve."24".Input.ManualOn )
   END_RUNG
   RUNG wire#powerrail
      Contact( #Tmp_EnableOperation )
      Contact( "DB_R134a_1_StepData"."Step"["DB_R134a_1_StepData".Values.CurrentStep].Valve[24] )
      Contact( "DB_R134a_BU_Values".Supply_AC.Output.FillUpCentralSupply )
      Coil( "DB_R134a_BU_Values".Valve."24".Input.AutoOn )
   END_RUNG
   RUNG wire#powerrail
      I_Contact( "DB_ALARM"."+KM1".CycleFault_38_A1 )
      I_Contact( "DB_ALARM"."+KM1".FillPressR134a.WireBreak )
      I_Contact( "DB_ALARM"."+KM1".FillPressR134a.FillUp )
      I_Contact( "DB_ALARM"."+KM1".FillPressR134a.MaxMax )
      Coil( "DB_R134a_BU_Values".Valve."24".Input.Release )
   END_RUNG
   RUNG wire#powerrail
      Coil( "DB_R134a_BU_Values".Valve."24".Input.SafetyRelease )
   END_RUNG
   RUNG wire#powerrail
      MOVE_BLK_VARIANT(SRC := "DB_R134a_1_StepData".Valve[24].Language, COUNT := 4, SRC_INDEX := 0, DEST_INDEX := 0, Ret_Val => #Tmp_ReturnValue, DEST => "DB_R134a_BU_Values".Valve."24".Input.TextName_Language)
   END_RUNG
   // the same network as SCL:
   "DB_R134a_BU_Values".Valve."24".Input.OpModeOutput := 0;
   "DB_R134a_BU_Values".Valve."24".Input.OpModeAutoManual := "DB_R134a_AT_2_Values".OperationMode.ManualValveControl;
   IF "DB_R134a_BU_Values".Valve."24".Input.OpModeAutoManual = 0 THEN
       "DB_R134a_BU_Values".Valve."24".Input.ManualOn := FALSE;
   END_IF;
   "DB_R134a_BU_Values".Valve."24".Input.AutoOn := #Tmp_EnableOperation AND "DB_R134a_1_StepData"."Step"["DB_R134a_1_StepData".Values.CurrentStep].Valve[24] AND "DB_R134a_BU_Values".Supply_AC.Output.FillUpCentralSupply;
   "DB_R134a_BU_Values".Valve."24".Input.Release := NOT "DB_ALARM"."+KM1".CycleFault_38_A1 AND NOT "DB_ALARM"."+KM1".FillPressR134a.WireBreak AND NOT "DB_ALARM"."+KM1".FillPressR134a.FillUp AND NOT "DB_ALARM"."+KM1".FillPressR134a.MaxMax;
   "DB_R134a_BU_Values".Valve."24".Input.SafetyRelease := TRUE;
   #Tmp_ReturnValue := MOVE_BLK_VARIANT(SRC := "DB_R134a_1_StepData".Valve[24].Language,
                           COUNT := 4,
                           SRC_INDEX := 0,
                           DEST_INDEX := 0,
                           DEST => "DB_R134a_BU_Values".Valve."24".Input.TextName_Language);
END_REGION

REGION Network 25: [24] valve 1KM1VI1KKP2KK21 - 100.21.3 - Supply central redundant // Versorgung - zentral - redundant
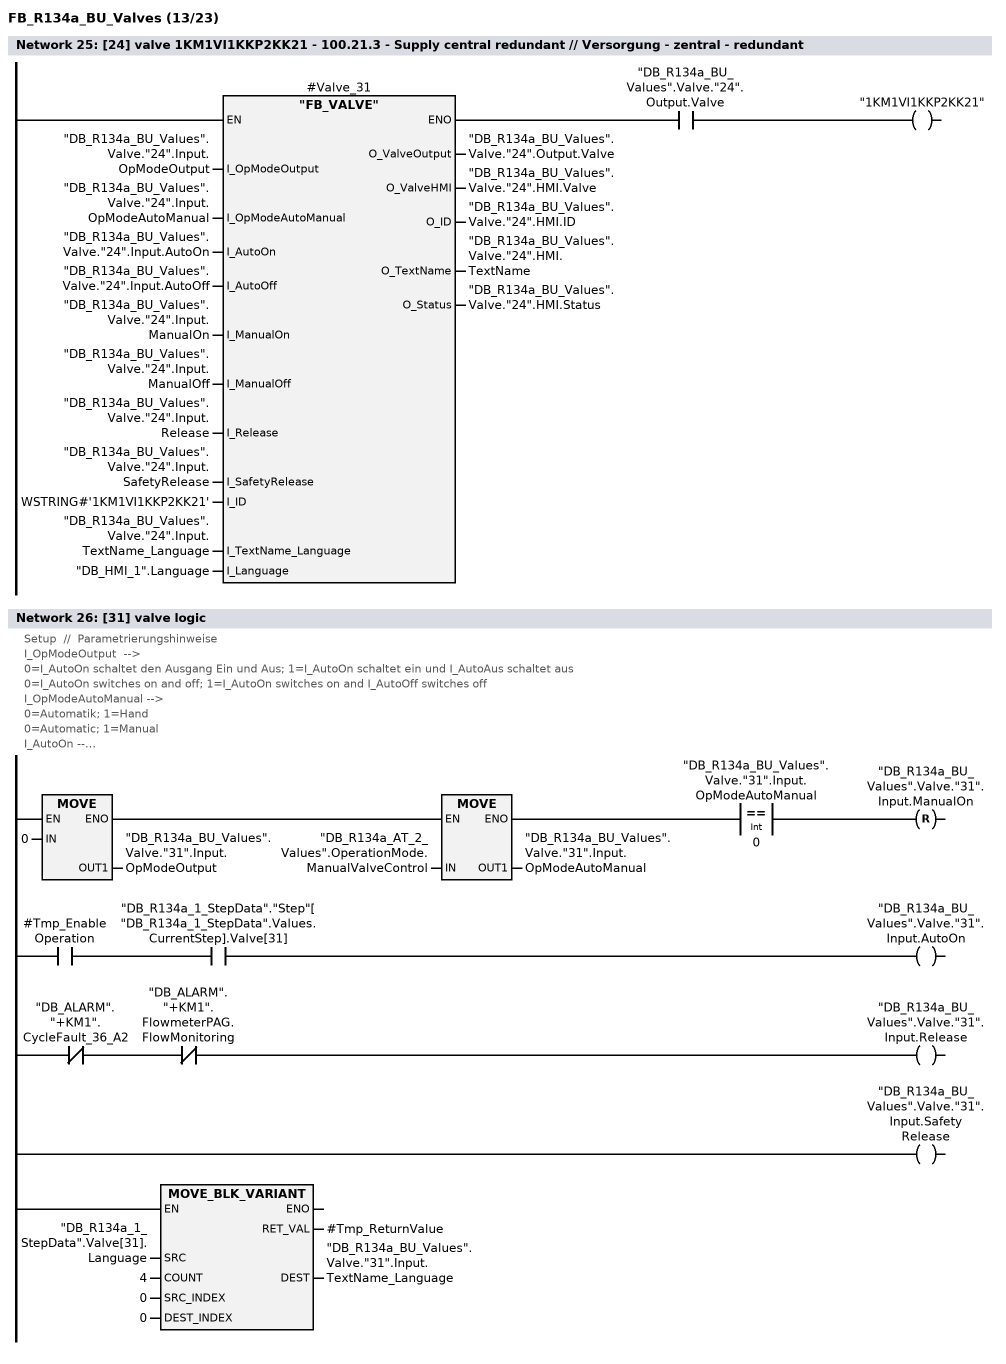
   RUNG wire#powerrail
      #Valve_31(I_OpModeOutput := "DB_R134a_BU_Values".Valve."24".Input.OpModeOutput, I_OpModeAutoManual := "DB_R134a_BU_Values".Valve."24".Input.OpModeAutoManual, I_AutoOn := "DB_R134a_BU_Values".Valve."24".Input.AutoOn, I_AutoOff := "DB_R134a_BU_Values".Valve."24".Input.AutoOff, I_ManualOn := "DB_R134a_BU_Values".Valve."24".Input.ManualOn, I_ManualOff := "DB_R134a_BU_Values".Valve."24".Input.ManualOff, I_Release := "DB_R134a_BU_Values".Valve."24".Input.Release, I_SafetyRelease := "DB_R134a_BU_Values".Valve."24".Input.SafetyRelease, I_ID := WSTRING#'1KM1VI1KKP2KK21', I_TextName_Language := "DB_R134a_BU_Values".Valve."24".Input.TextName_Language, I_Language := "DB_HMI_1".Language, O_ValveOutput => "DB_R134a_BU_Values".Valve."24".Output.Valve, O_ValveHMI => "DB_R134a_BU_Values".Valve."24".HMI.Valve, O_ID => "DB_R134a_BU_Values".Valve."24".HMI.ID, O_TextName => "DB_R134a_BU_Values".Valve."24".HMI.TextName, O_Status => "DB_R134a_BU_Values".Valve."24".HMI.Status)
      Contact( "DB_R134a_BU_Values".Valve."24".Output.Valve )
      Coil( "1KM1VI1KKP2KK21" )
   END_RUNG
   // the same network as SCL:
   #Valve_31(I_OpModeOutput := "DB_R134a_BU_Values".Valve."24".Input.OpModeOutput,   // "FB_VALVE"
             I_OpModeAutoManual := "DB_R134a_BU_Values".Valve."24".Input.OpModeAutoManual,
             I_AutoOn := "DB_R134a_BU_Values".Valve."24".Input.AutoOn,
             I_AutoOff := "DB_R134a_BU_Values".Valve."24".Input.AutoOff,
             I_ManualOn := "DB_R134a_BU_Values".Valve."24".Input.ManualOn,
             I_ManualOff := "DB_R134a_BU_Values".Valve."24".Input.ManualOff,
             I_Release := "DB_R134a_BU_Values".Valve."24".Input.Release,
             I_SafetyRelease := "DB_R134a_BU_Values".Valve."24".Input.SafetyRelease,
             I_ID := WSTRING#'1KM1VI1KKP2KK21',
             I_TextName_Language := "DB_R134a_BU_Values".Valve."24".Input.TextName_Language,
             I_Language := "DB_HMI_1".Language,
             O_ValveOutput => "DB_R134a_BU_Values".Valve."24".Output.Valve,
             O_ValveHMI => "DB_R134a_BU_Values".Valve."24".HMI.Valve,
             O_ID => "DB_R134a_BU_Values".Valve."24".HMI.ID,
             O_TextName => "DB_R134a_BU_Values".Valve."24".HMI.TextName,
             O_Status => "DB_R134a_BU_Values".Valve."24".HMI.Status,
             ENO => #_w1);
   "1KM1VI1KKP2KK21" := #_w1 AND "DB_R134a_BU_Values".Valve."24".Output.Valve;
END_REGION

REGION Network 26: [31] valve logic
   // Setup  //  Parametrierungshinweise
   // I_OpModeOutput  -->
   // 0=I_AutoOn schaltet den Ausgang Ein und Aus; 1=I_AutoOn schaltet ein und I_AutoAus schaltet aus
   // 0=I_AutoOn switches on and off; 1=I_AutoOn switches on and I_AutoOff switches off
   // 
   // I_OpModeAutoManual -->
   // 0=Automatik; 1=Hand
   // 0=Automatic; 1=Manual
   // 
   // I_AutoOn -->
   // 1=Automatik Ein, Eingang für die normalen Ventilverschaltungsbedingungen
   // 1=Automatic On, Input for the normal valve conditions
   // 
   // I_Release -->
   // 1=Freigabe, Eingang für die Fehlerbedingungen
   // 1=Release, Input for fault conditions
   // 
   // I_SafetyRelease -->
   // 1=Sicherheitsfreigabe, Eingang für zusätzliche Schaltbefehle aus dem Sicherheitsprogramm
   // 1=Safety release, Input for additional safety conditions from the safety program
   RUNG wire#powerrail
      Move(in := 0, out1 => "DB_R134a_BU_Values".Valve."31".Input.OpModeOutput)
      Move(in := "DB_R134a_AT_2_Values".OperationMode.ManualValveControl, out1 => "DB_R134a_BU_Values".Valve."31".Input.OpModeAutoManual)
      { S7_Templates := "SrcType := Int" } EQ_Contact(in1 := "DB_R134a_BU_Values".Valve."31".Input.OpModeAutoManual, in2 := 0)
      R_Coil( "DB_R134a_BU_Values".Valve."31".Input.ManualOn )
   END_RUNG
   RUNG wire#powerrail
      Contact( #Tmp_EnableOperation )
      Contact( "DB_R134a_1_StepData"."Step"["DB_R134a_1_StepData".Values.CurrentStep].Valve[31] )
      Coil( "DB_R134a_BU_Values".Valve."31".Input.AutoOn )
   END_RUNG
   RUNG wire#powerrail
      I_Contact( "DB_ALARM"."+KM1".CycleFault_36_A2 )
      I_Contact( "DB_ALARM"."+KM1".FlowmeterPAG.FlowMonitoring )
      Coil( "DB_R134a_BU_Values".Valve."31".Input.Release )
   END_RUNG
   RUNG wire#powerrail
      Coil( "DB_R134a_BU_Values".Valve."31".Input.SafetyRelease )
   END_RUNG
   RUNG wire#powerrail
      MOVE_BLK_VARIANT(SRC := "DB_R134a_1_StepData".Valve[31].Language, COUNT := 4, SRC_INDEX := 0, DEST_INDEX := 0, Ret_Val => #Tmp_ReturnValue, DEST => "DB_R134a_BU_Values".Valve."31".Input.TextName_Language)
   END_RUNG
   // the same network as SCL:
   "DB_R134a_BU_Values".Valve."31".Input.OpModeOutput := 0;
   "DB_R134a_BU_Values".Valve."31".Input.OpModeAutoManual := "DB_R134a_AT_2_Values".OperationMode.ManualValveControl;
   IF "DB_R134a_BU_Values".Valve."31".Input.OpModeAutoManual = 0 THEN
       "DB_R134a_BU_Values".Valve."31".Input.ManualOn := FALSE;
   END_IF;
   "DB_R134a_BU_Values".Valve."31".Input.AutoOn := #Tmp_EnableOperation AND "DB_R134a_1_StepData"."Step"["DB_R134a_1_StepData".Values.CurrentStep].Valve[31];
   "DB_R134a_BU_Values".Valve."31".Input.Release := NOT "DB_ALARM"."+KM1".CycleFault_36_A2 AND NOT "DB_ALARM"."+KM1".FlowmeterPAG.FlowMonitoring;
   "DB_R134a_BU_Values".Valve."31".Input.SafetyRelease := TRUE;
   #Tmp_ReturnValue := MOVE_BLK_VARIANT(SRC := "DB_R134a_1_StepData".Valve[31].Language,
                           COUNT := 4,
                           SRC_INDEX := 0,
                           DEST_INDEX := 0,
                           DEST => "DB_R134a_BU_Values".Valve."31".Input.TextName_Language);
END_REGION

REGION Network 27: [31] valve 1KM1VI1KKP9KK102 - 108.102.6 - filling before adapter PAG // Füllen vor Adapter PAG
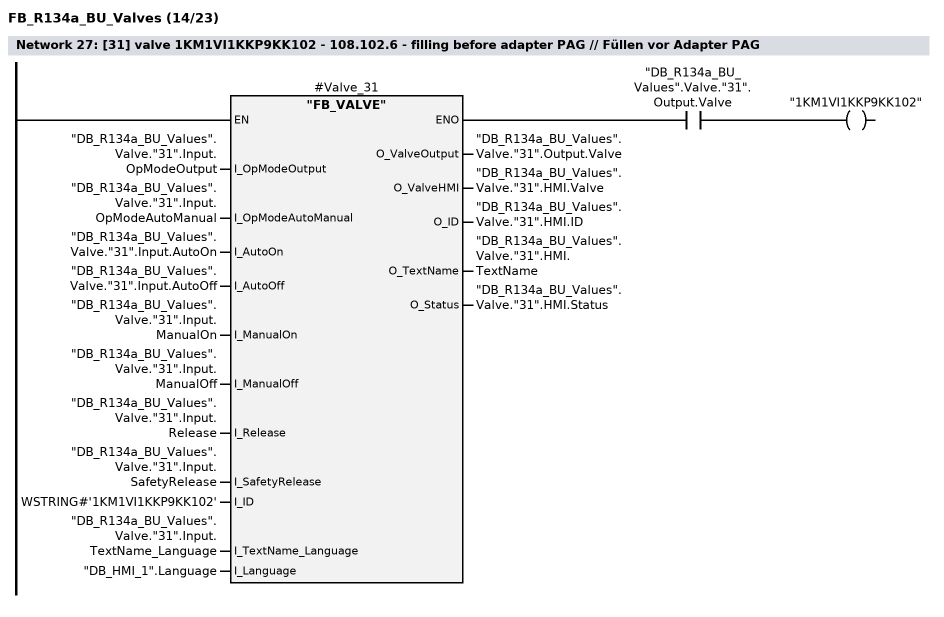
   RUNG wire#powerrail
      #Valve_31(I_OpModeOutput := "DB_R134a_BU_Values".Valve."31".Input.OpModeOutput, I_OpModeAutoManual := "DB_R134a_BU_Values".Valve."31".Input.OpModeAutoManual, I_AutoOn := "DB_R134a_BU_Values".Valve."31".Input.AutoOn, I_AutoOff := "DB_R134a_BU_Values".Valve."31".Input.AutoOff, I_ManualOn := "DB_R134a_BU_Values".Valve."31".Input.ManualOn, I_ManualOff := "DB_R134a_BU_Values".Valve."31".Input.ManualOff, I_Release := "DB_R134a_BU_Values".Valve."31".Input.Release, I_SafetyRelease := "DB_R134a_BU_Values".Valve."31".Input.SafetyRelease, I_ID := WSTRING#'1KM1VI1KKP9KK102', I_TextName_Language := "DB_R134a_BU_Values".Valve."31".Input.TextName_Language, I_Language := "DB_HMI_1".Language, O_ValveOutput => "DB_R134a_BU_Values".Valve."31".Output.Valve, O_ValveHMI => "DB_R134a_BU_Values".Valve."31".HMI.Valve, O_ID => "DB_R134a_BU_Values".Valve."31".HMI.ID, O_TextName => "DB_R134a_BU_Values".Valve."31".HMI.TextName, O_Status => "DB_R134a_BU_Values".Valve."31".HMI.Status)
      Contact( "DB_R134a_BU_Values".Valve."31".Output.Valve )
      Coil( "1KM1VI1KKP9KK102" )
   END_RUNG
   // the same network as SCL:
   #Valve_31(I_OpModeOutput := "DB_R134a_BU_Values".Valve."31".Input.OpModeOutput,   // "FB_VALVE"
             I_OpModeAutoManual := "DB_R134a_BU_Values".Valve."31".Input.OpModeAutoManual,
             I_AutoOn := "DB_R134a_BU_Values".Valve."31".Input.AutoOn,
             I_AutoOff := "DB_R134a_BU_Values".Valve."31".Input.AutoOff,
             I_ManualOn := "DB_R134a_BU_Values".Valve."31".Input.ManualOn,
             I_ManualOff := "DB_R134a_BU_Values".Valve."31".Input.ManualOff,
             I_Release := "DB_R134a_BU_Values".Valve."31".Input.Release,
             I_SafetyRelease := "DB_R134a_BU_Values".Valve."31".Input.SafetyRelease,
             I_ID := WSTRING#'1KM1VI1KKP9KK102',
             I_TextName_Language := "DB_R134a_BU_Values".Valve."31".Input.TextName_Language,
             I_Language := "DB_HMI_1".Language,
             O_ValveOutput => "DB_R134a_BU_Values".Valve."31".Output.Valve,
             O_ValveHMI => "DB_R134a_BU_Values".Valve."31".HMI.Valve,
             O_ID => "DB_R134a_BU_Values".Valve."31".HMI.ID,
             O_TextName => "DB_R134a_BU_Values".Valve."31".HMI.TextName,
             O_Status => "DB_R134a_BU_Values".Valve."31".HMI.Status,
             ENO => #_w1);
   "1KM1VI1KKP9KK102" := #_w1 AND "DB_R134a_BU_Values".Valve."31".Output.Valve;
END_REGION

REGION Network 28: [43] valve logic
   // Setup  //  Parametrierungshinweise
   // I_OpModeOutput  -->
   // 0=I_AutoOn schaltet den Ausgang Ein und Aus; 1=I_AutoOn schaltet ein und I_AutoAus schaltet aus
   // 0=I_AutoOn switches on and off; 1=I_AutoOn switches on and I_AutoOff switches off
   // 
   // I_OpModeAutoManual -->
   // 0=Automatik; 1=Hand
   // 0=Automatic; 1=Manual
   // 
   // I_AutoOn -->
   // 1=Automatik Ein, Eingang für die normalen Ventilverschaltungsbedingungen
   // 1=Automatic On, Input for the normal valve conditions
   // 
   // I_Release -->
   // 1=Freigabe, Eingang für die Fehlerbedingungen
   // 1=Release, Input for fault conditions
   // 
   // I_SafetyRelease -->
   // 1=Sicherheitsfreigabe, Eingang für zusätzliche Schaltbefehle aus dem Sicherheitsprogramm
   // 1=Safety release, Input for additional safety conditions from the safety program
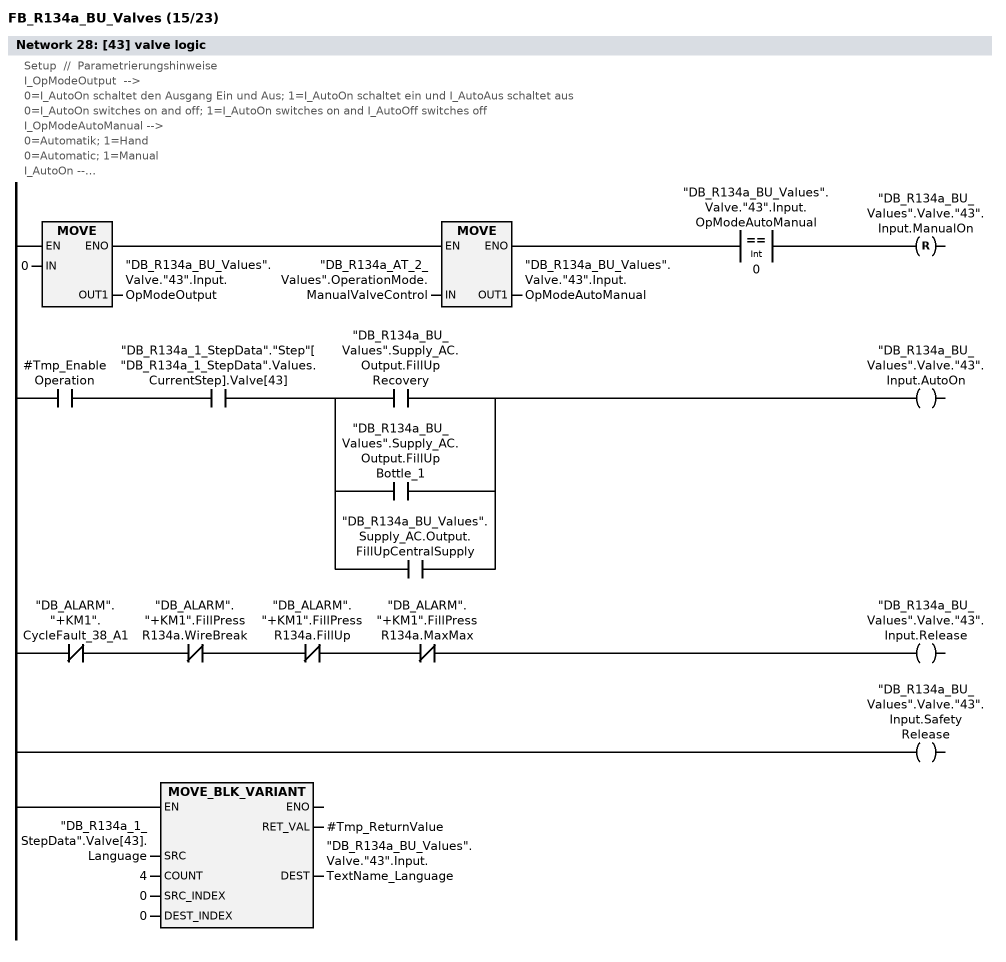
   RUNG wire#powerrail
      Move(in := 0, out1 => "DB_R134a_BU_Values".Valve."43".Input.OpModeOutput)
      Move(in := "DB_R134a_AT_2_Values".OperationMode.ManualValveControl, out1 => "DB_R134a_BU_Values".Valve."43".Input.OpModeAutoManual)
      { S7_Templates := "SrcType := Int" } EQ_Contact(in1 := "DB_R134a_BU_Values".Valve."43".Input.OpModeAutoManual, in2 := 0)
      R_Coil( "DB_R134a_BU_Values".Valve."43".Input.ManualOn )
   END_RUNG
   RUNG wire#powerrail
      Contact( #Tmp_EnableOperation )
      Contact( "DB_R134a_1_StepData"."Step"["DB_R134a_1_StepData".Values.CurrentStep].Valve[43] )
      wire#w1
      Contact( "DB_R134a_BU_Values".Supply_AC.Output.FillUpRecovery )
      wire#w2
      Coil( "DB_R134a_BU_Values".Valve."43".Input.AutoOn )
   END_RUNG
   RUNG wire#w1
      Contact( "DB_R134a_BU_Values".Supply_AC.Output.FillUpBottle_1 )
   END_RUNG wire#w2
   RUNG wire#w1
      Contact( "DB_R134a_BU_Values".Supply_AC.Output.FillUpCentralSupply )
   END_RUNG wire#w2
   RUNG wire#powerrail
      I_Contact( "DB_ALARM"."+KM1".CycleFault_38_A1 )
      I_Contact( "DB_ALARM"."+KM1".FillPressR134a.WireBreak )
      I_Contact( "DB_ALARM"."+KM1".FillPressR134a.FillUp )
      I_Contact( "DB_ALARM"."+KM1".FillPressR134a.MaxMax )
      Coil( "DB_R134a_BU_Values".Valve."43".Input.Release )
   END_RUNG
   RUNG wire#powerrail
      Coil( "DB_R134a_BU_Values".Valve."43".Input.SafetyRelease )
   END_RUNG
   RUNG wire#powerrail
      MOVE_BLK_VARIANT(SRC := "DB_R134a_1_StepData".Valve[43].Language, COUNT := 4, SRC_INDEX := 0, DEST_INDEX := 0, Ret_Val => #Tmp_ReturnValue, DEST => "DB_R134a_BU_Values".Valve."43".Input.TextName_Language)
   END_RUNG
   // the same network as SCL:
   "DB_R134a_BU_Values".Valve."43".Input.OpModeOutput := 0;
   "DB_R134a_BU_Values".Valve."43".Input.OpModeAutoManual := "DB_R134a_AT_2_Values".OperationMode.ManualValveControl;
   IF "DB_R134a_BU_Values".Valve."43".Input.OpModeAutoManual = 0 THEN
       "DB_R134a_BU_Values".Valve."43".Input.ManualOn := FALSE;
   END_IF;
   "DB_R134a_BU_Values".Valve."43".Input.AutoOn := #Tmp_EnableOperation AND "DB_R134a_1_StepData"."Step"["DB_R134a_1_StepData".Values.CurrentStep].Valve[43] AND ("DB_R134a_BU_Values".Supply_AC.Output.FillUpRecovery OR "DB_R134a_BU_Values".Supply_AC.Output.FillUpBottle_1 OR "DB_R134a_BU_Values".Supply_AC.Output.FillUpCentralSupply);
   "DB_R134a_BU_Values".Valve."43".Input.Release := NOT "DB_ALARM"."+KM1".CycleFault_38_A1 AND NOT "DB_ALARM"."+KM1".FillPressR134a.WireBreak AND NOT "DB_ALARM"."+KM1".FillPressR134a.FillUp AND NOT "DB_ALARM"."+KM1".FillPressR134a.MaxMax;
   "DB_R134a_BU_Values".Valve."43".Input.SafetyRelease := TRUE;
   #Tmp_ReturnValue := MOVE_BLK_VARIANT(SRC := "DB_R134a_1_StepData".Valve[43].Language,
                           COUNT := 4,
                           SRC_INDEX := 0,
                           DEST_INDEX := 0,
                           DEST => "DB_R134a_BU_Values".Valve."43".Input.TextName_Language);
END_REGION

REGION Network 29: [43] valve 1KM1VI1KKP1KK101 - 100.101.3 - filling entry R134a // Füllen Eintritt R134a Speicher
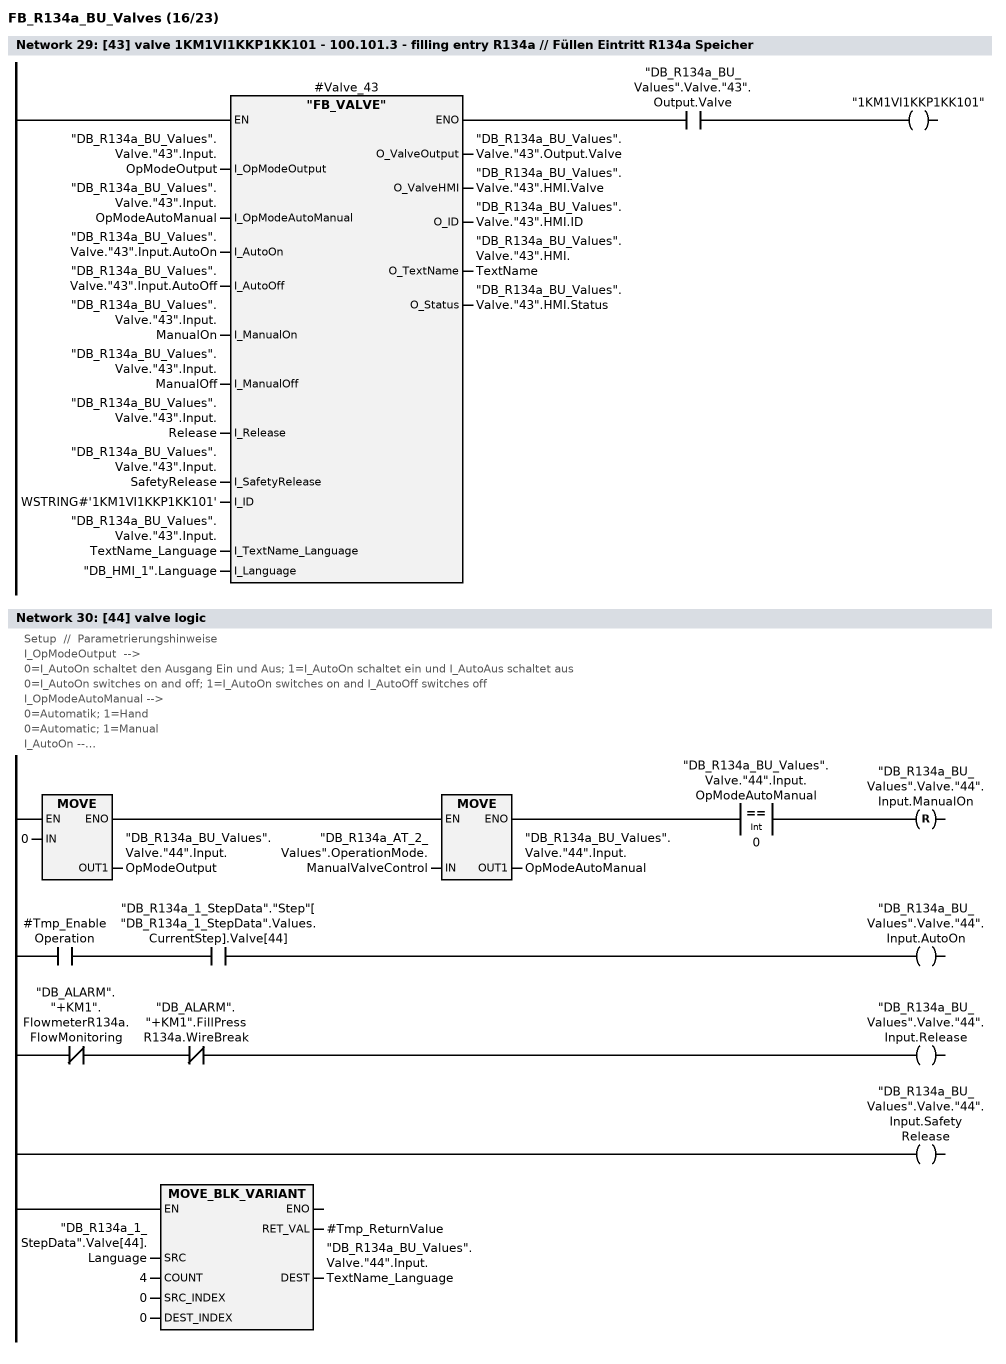
   RUNG wire#powerrail
      #Valve_43(I_OpModeOutput := "DB_R134a_BU_Values".Valve."43".Input.OpModeOutput, I_OpModeAutoManual := "DB_R134a_BU_Values".Valve."43".Input.OpModeAutoManual, I_AutoOn := "DB_R134a_BU_Values".Valve."43".Input.AutoOn, I_AutoOff := "DB_R134a_BU_Values".Valve."43".Input.AutoOff, I_ManualOn := "DB_R134a_BU_Values".Valve."43".Input.ManualOn, I_ManualOff := "DB_R134a_BU_Values".Valve."43".Input.ManualOff, I_Release := "DB_R134a_BU_Values".Valve."43".Input.Release, I_SafetyRelease := "DB_R134a_BU_Values".Valve."43".Input.SafetyRelease, I_ID := WSTRING#'1KM1VI1KKP1KK101', I_TextName_Language := "DB_R134a_BU_Values".Valve."43".Input.TextName_Language, I_Language := "DB_HMI_1".Language, O_ValveOutput => "DB_R134a_BU_Values".Valve."43".Output.Valve, O_ValveHMI => "DB_R134a_BU_Values".Valve."43".HMI.Valve, O_ID => "DB_R134a_BU_Values".Valve."43".HMI.ID, O_TextName => "DB_R134a_BU_Values".Valve."43".HMI.TextName, O_Status => "DB_R134a_BU_Values".Valve."43".HMI.Status)
      Contact( "DB_R134a_BU_Values".Valve."43".Output.Valve )
      Coil( "1KM1VI1KKP1KK101" )
   END_RUNG
   // the same network as SCL:
   #Valve_43(I_OpModeOutput := "DB_R134a_BU_Values".Valve."43".Input.OpModeOutput,   // "FB_VALVE"
             I_OpModeAutoManual := "DB_R134a_BU_Values".Valve."43".Input.OpModeAutoManual,
             I_AutoOn := "DB_R134a_BU_Values".Valve."43".Input.AutoOn,
             I_AutoOff := "DB_R134a_BU_Values".Valve."43".Input.AutoOff,
             I_ManualOn := "DB_R134a_BU_Values".Valve."43".Input.ManualOn,
             I_ManualOff := "DB_R134a_BU_Values".Valve."43".Input.ManualOff,
             I_Release := "DB_R134a_BU_Values".Valve."43".Input.Release,
             I_SafetyRelease := "DB_R134a_BU_Values".Valve."43".Input.SafetyRelease,
             I_ID := WSTRING#'1KM1VI1KKP1KK101',
             I_TextName_Language := "DB_R134a_BU_Values".Valve."43".Input.TextName_Language,
             I_Language := "DB_HMI_1".Language,
             O_ValveOutput => "DB_R134a_BU_Values".Valve."43".Output.Valve,
             O_ValveHMI => "DB_R134a_BU_Values".Valve."43".HMI.Valve,
             O_ID => "DB_R134a_BU_Values".Valve."43".HMI.ID,
             O_TextName => "DB_R134a_BU_Values".Valve."43".HMI.TextName,
             O_Status => "DB_R134a_BU_Values".Valve."43".HMI.Status,
             ENO => #_w1);
   "1KM1VI1KKP1KK101" := #_w1 AND "DB_R134a_BU_Values".Valve."43".Output.Valve;
END_REGION

REGION Network 30: [44] valve logic
   // Setup  //  Parametrierungshinweise
   // I_OpModeOutput  -->
   // 0=I_AutoOn schaltet den Ausgang Ein und Aus; 1=I_AutoOn schaltet ein und I_AutoAus schaltet aus
   // 0=I_AutoOn switches on and off; 1=I_AutoOn switches on and I_AutoOff switches off
   // 
   // I_OpModeAutoManual -->
   // 0=Automatik; 1=Hand
   // 0=Automatic; 1=Manual
   // 
   // I_AutoOn -->
   // 1=Automatik Ein, Eingang für die normalen Ventilverschaltungsbedingungen
   // 1=Automatic On, Input for the normal valve conditions
   // 
   // I_Release -->
   // 1=Freigabe, Eingang für die Fehlerbedingungen
   // 1=Release, Input for fault conditions
   // 
   // I_SafetyRelease -->
   // 1=Sicherheitsfreigabe, Eingang für zusätzliche Schaltbefehle aus dem Sicherheitsprogramm
   // 1=Safety release, Input for additional safety conditions from the safety program
   RUNG wire#powerrail
      Move(in := 0, out1 => "DB_R134a_BU_Values".Valve."44".Input.OpModeOutput)
      Move(in := "DB_R134a_AT_2_Values".OperationMode.ManualValveControl, out1 => "DB_R134a_BU_Values".Valve."44".Input.OpModeAutoManual)
      { S7_Templates := "SrcType := Int" } EQ_Contact(in1 := "DB_R134a_BU_Values".Valve."44".Input.OpModeAutoManual, in2 := 0)
      R_Coil( "DB_R134a_BU_Values".Valve."44".Input.ManualOn )
   END_RUNG
   RUNG wire#powerrail
      Contact( #Tmp_EnableOperation )
      Contact( "DB_R134a_1_StepData"."Step"["DB_R134a_1_StepData".Values.CurrentStep].Valve[44] )
      Coil( "DB_R134a_BU_Values".Valve."44".Input.AutoOn )
   END_RUNG
   RUNG wire#powerrail
      I_Contact( "DB_ALARM"."+KM1".FlowmeterR134a.FlowMonitoring )
      I_Contact( "DB_ALARM"."+KM1".FillPressR134a.WireBreak )
      Coil( "DB_R134a_BU_Values".Valve."44".Input.Release )
   END_RUNG
   RUNG wire#powerrail
      Coil( "DB_R134a_BU_Values".Valve."44".Input.SafetyRelease )
   END_RUNG
   RUNG wire#powerrail
      MOVE_BLK_VARIANT(SRC := "DB_R134a_1_StepData".Valve[44].Language, COUNT := 4, SRC_INDEX := 0, DEST_INDEX := 0, Ret_Val => #Tmp_ReturnValue, DEST => "DB_R134a_BU_Values".Valve."44".Input.TextName_Language)
   END_RUNG
   // the same network as SCL:
   "DB_R134a_BU_Values".Valve."44".Input.OpModeOutput := 0;
   "DB_R134a_BU_Values".Valve."44".Input.OpModeAutoManual := "DB_R134a_AT_2_Values".OperationMode.ManualValveControl;
   IF "DB_R134a_BU_Values".Valve."44".Input.OpModeAutoManual = 0 THEN
       "DB_R134a_BU_Values".Valve."44".Input.ManualOn := FALSE;
   END_IF;
   "DB_R134a_BU_Values".Valve."44".Input.AutoOn := #Tmp_EnableOperation AND "DB_R134a_1_StepData"."Step"["DB_R134a_1_StepData".Values.CurrentStep].Valve[44];
   "DB_R134a_BU_Values".Valve."44".Input.Release := NOT "DB_ALARM"."+KM1".FlowmeterR134a.FlowMonitoring AND NOT "DB_ALARM"."+KM1".FillPressR134a.WireBreak;
   "DB_R134a_BU_Values".Valve."44".Input.SafetyRelease := TRUE;
   #Tmp_ReturnValue := MOVE_BLK_VARIANT(SRC := "DB_R134a_1_StepData".Valve[44].Language,
                           COUNT := 4,
                           SRC_INDEX := 0,
                           DEST_INDEX := 0,
                           DEST => "DB_R134a_BU_Values".Valve."44".Input.TextName_Language);
END_REGION

REGION Network 31: [44] valve 1KM1VI1KKP1KK101 - 100.102.3 - filling before adapter R134a // Füllen vor Adapter R134a
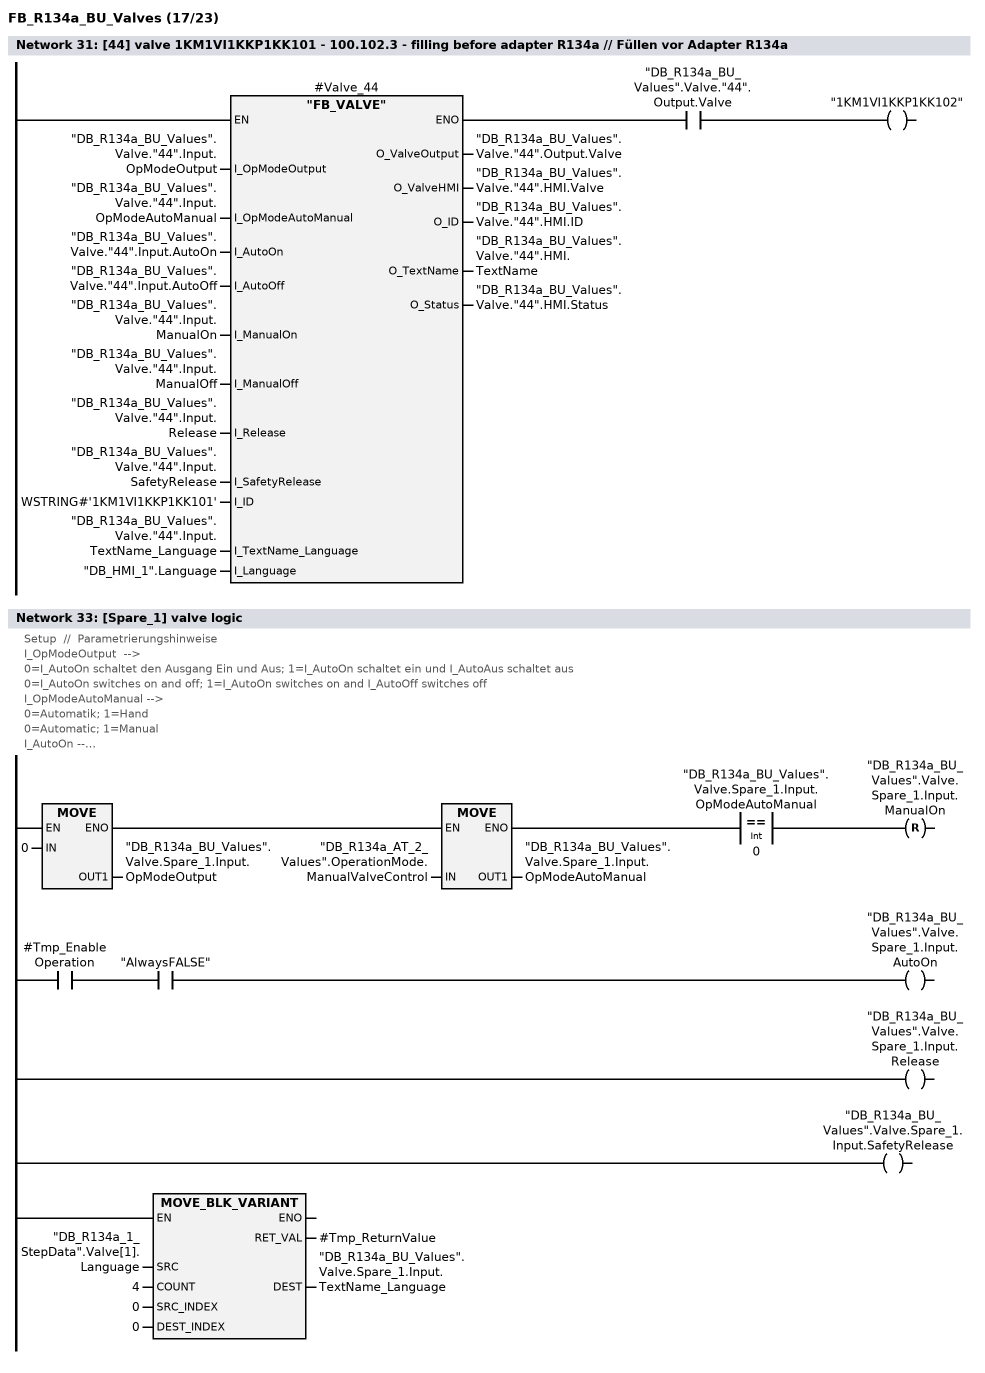
   RUNG wire#powerrail
      #Valve_44(I_OpModeOutput := "DB_R134a_BU_Values".Valve."44".Input.OpModeOutput, I_OpModeAutoManual := "DB_R134a_BU_Values".Valve."44".Input.OpModeAutoManual, I_AutoOn := "DB_R134a_BU_Values".Valve."44".Input.AutoOn, I_AutoOff := "DB_R134a_BU_Values".Valve."44".Input.AutoOff, I_ManualOn := "DB_R134a_BU_Values".Valve."44".Input.ManualOn, I_ManualOff := "DB_R134a_BU_Values".Valve."44".Input.ManualOff, I_Release := "DB_R134a_BU_Values".Valve."44".Input.Release, I_SafetyRelease := "DB_R134a_BU_Values".Valve."44".Input.SafetyRelease, I_ID := WSTRING#'1KM1VI1KKP1KK101', I_TextName_Language := "DB_R134a_BU_Values".Valve."44".Input.TextName_Language, I_Language := "DB_HMI_1".Language, O_ValveOutput => "DB_R134a_BU_Values".Valve."44".Output.Valve, O_ValveHMI => "DB_R134a_BU_Values".Valve."44".HMI.Valve, O_ID => "DB_R134a_BU_Values".Valve."44".HMI.ID, O_TextName => "DB_R134a_BU_Values".Valve."44".HMI.TextName, O_Status => "DB_R134a_BU_Values".Valve."44".HMI.Status)
      Contact( "DB_R134a_BU_Values".Valve."44".Output.Valve )
      Coil( "1KM1VI1KKP1KK102" )
   END_RUNG
   // the same network as SCL:
   #Valve_44(I_OpModeOutput := "DB_R134a_BU_Values".Valve."44".Input.OpModeOutput,   // "FB_VALVE"
             I_OpModeAutoManual := "DB_R134a_BU_Values".Valve."44".Input.OpModeAutoManual,
             I_AutoOn := "DB_R134a_BU_Values".Valve."44".Input.AutoOn,
             I_AutoOff := "DB_R134a_BU_Values".Valve."44".Input.AutoOff,
             I_ManualOn := "DB_R134a_BU_Values".Valve."44".Input.ManualOn,
             I_ManualOff := "DB_R134a_BU_Values".Valve."44".Input.ManualOff,
             I_Release := "DB_R134a_BU_Values".Valve."44".Input.Release,
             I_SafetyRelease := "DB_R134a_BU_Values".Valve."44".Input.SafetyRelease,
             I_ID := WSTRING#'1KM1VI1KKP1KK101',
             I_TextName_Language := "DB_R134a_BU_Values".Valve."44".Input.TextName_Language,
             I_Language := "DB_HMI_1".Language,
             O_ValveOutput => "DB_R134a_BU_Values".Valve."44".Output.Valve,
             O_ValveHMI => "DB_R134a_BU_Values".Valve."44".HMI.Valve,
             O_ID => "DB_R134a_BU_Values".Valve."44".HMI.ID,
             O_TextName => "DB_R134a_BU_Values".Valve."44".HMI.TextName,
             O_Status => "DB_R134a_BU_Values".Valve."44".HMI.Status,
             ENO => #_w1);
   "1KM1VI1KKP1KK102" := #_w1 AND "DB_R134a_BU_Values".Valve."44".Output.Valve;
END_REGION

REGION Network 32: ------------- Valves spare -------------
   // This network is only here to make the PLC program more structured/readable // Dieses Netzwerk ist nur hier um die Lesbarkeit des SPS-Programms zu erhöhen
END_REGION

REGION Network 33: [Spare_1] valve logic
   // Setup  //  Parametrierungshinweise
   // I_OpModeOutput  -->
   // 0=I_AutoOn schaltet den Ausgang Ein und Aus; 1=I_AutoOn schaltet ein und I_AutoAus schaltet aus
   // 0=I_AutoOn switches on and off; 1=I_AutoOn switches on and I_AutoOff switches off
   // 
   // I_OpModeAutoManual -->
   // 0=Automatik; 1=Hand
   // 0=Automatic; 1=Manual
   // 
   // I_AutoOn -->
   // 1=Automatik Ein, Eingang für die normalen Ventilverschaltungsbedingungen
   // 1=Automatic On, Input for the normal valve conditions
   // 
   // I_Release -->
   // 1=Freigabe, Eingang für die Fehlerbedingungen
   // 1=Release, Input for fault conditions
   // 
   // I_SafetyRelease -->
   // 1=Sicherheitsfreigabe, Eingang für zusätzliche Schaltbefehle aus dem Sicherheitsprogramm
   // 1=Safety release, Input for additional safety conditions from the safety program
   RUNG wire#powerrail
      Move(in := 0, out1 => "DB_R134a_BU_Values".Valve.Spare_1.Input.OpModeOutput)
      Move(in := "DB_R134a_AT_2_Values".OperationMode.ManualValveControl, out1 => "DB_R134a_BU_Values".Valve.Spare_1.Input.OpModeAutoManual)
      { S7_Templates := "SrcType := Int" } EQ_Contact(in1 := "DB_R134a_BU_Values".Valve.Spare_1.Input.OpModeAutoManual, in2 := 0)
      R_Coil( "DB_R134a_BU_Values".Valve.Spare_1.Input.ManualOn )
   END_RUNG
   RUNG wire#powerrail
      Contact( #Tmp_EnableOperation )
      Contact( "AlwaysFALSE" )
      Coil( "DB_R134a_BU_Values".Valve.Spare_1.Input.AutoOn )
   END_RUNG
   RUNG wire#powerrail
      Coil( "DB_R134a_BU_Values".Valve.Spare_1.Input.Release )
   END_RUNG
   RUNG wire#powerrail
      Coil( "DB_R134a_BU_Values".Valve.Spare_1.Input.SafetyRelease )
   END_RUNG
   RUNG wire#powerrail
      MOVE_BLK_VARIANT(SRC := "DB_R134a_1_StepData".Valve[1].Language, COUNT := 4, SRC_INDEX := 0, DEST_INDEX := 0, Ret_Val => #Tmp_ReturnValue, DEST => "DB_R134a_BU_Values".Valve.Spare_1.Input.TextName_Language)
   END_RUNG
   // the same network as SCL:
   "DB_R134a_BU_Values".Valve.Spare_1.Input.OpModeOutput := 0;
   "DB_R134a_BU_Values".Valve.Spare_1.Input.OpModeAutoManual := "DB_R134a_AT_2_Values".OperationMode.ManualValveControl;
   IF "DB_R134a_BU_Values".Valve.Spare_1.Input.OpModeAutoManual = 0 THEN
       "DB_R134a_BU_Values".Valve.Spare_1.Input.ManualOn := FALSE;
   END_IF;
   "DB_R134a_BU_Values".Valve.Spare_1.Input.AutoOn := #Tmp_EnableOperation AND "AlwaysFALSE";
   "DB_R134a_BU_Values".Valve.Spare_1.Input.Release := TRUE;
   "DB_R134a_BU_Values".Valve.Spare_1.Input.SafetyRelease := TRUE;
   #Tmp_ReturnValue := MOVE_BLK_VARIANT(SRC := "DB_R134a_1_StepData".Valve[1].Language,
                           COUNT := 4,
                           SRC_INDEX := 0,
                           DEST_INDEX := 0,
                           DEST => "DB_R134a_BU_Values".Valve.Spare_1.Input.TextName_Language);
END_REGION

REGION Network 34: [Spare_1] valve 1KM1VI1KKP10KKR14 - xxx.. - spare // Reserve
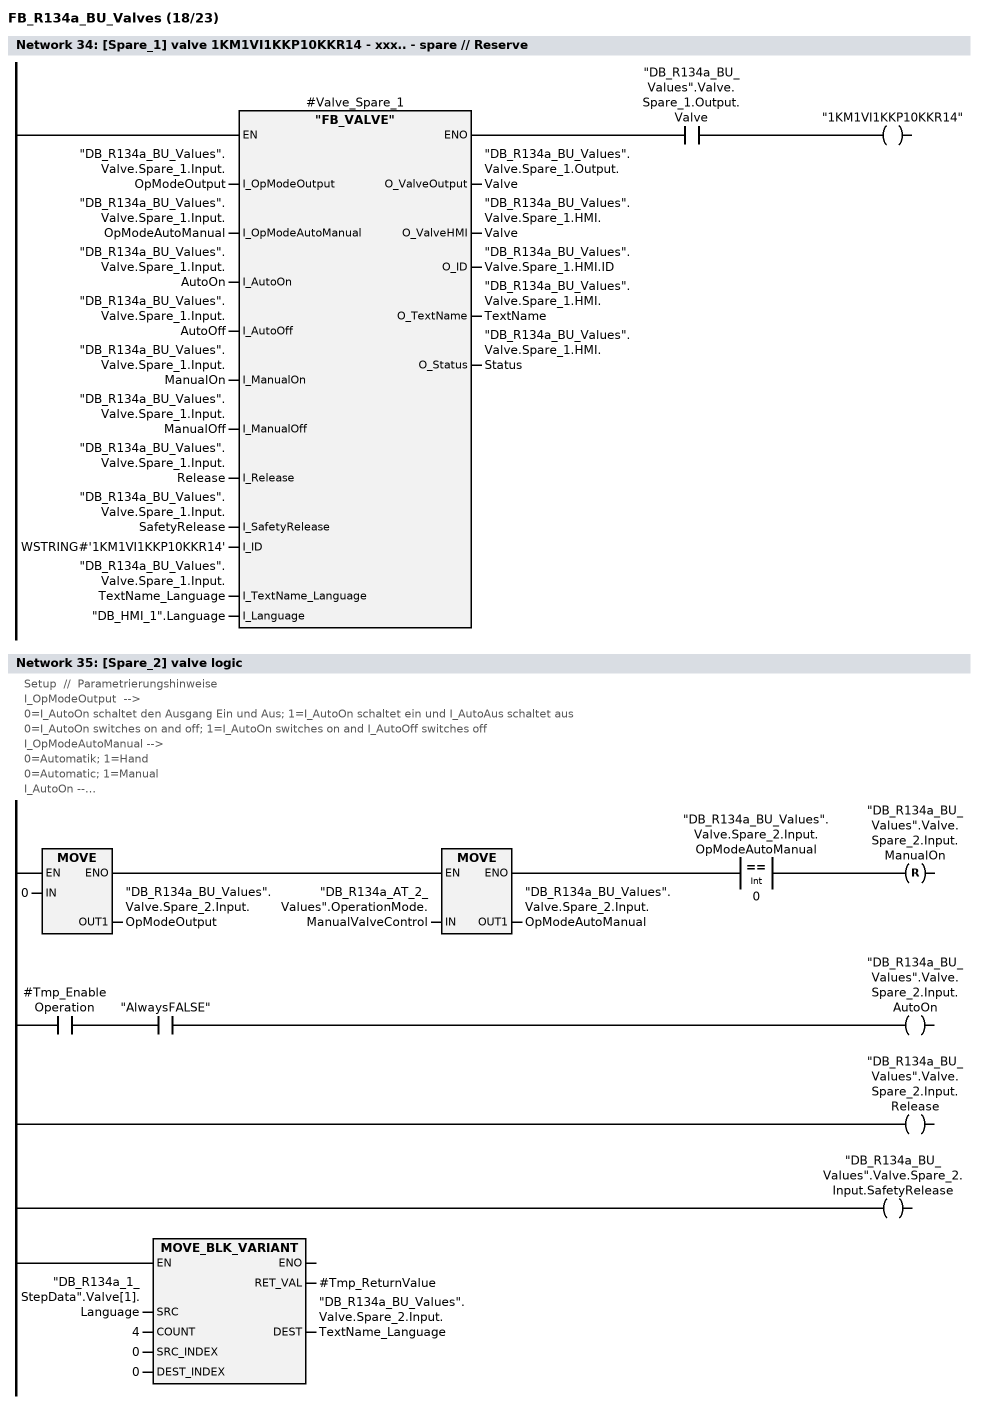
   RUNG wire#powerrail
      #Valve_Spare_1(I_OpModeOutput := "DB_R134a_BU_Values".Valve.Spare_1.Input.OpModeOutput, I_OpModeAutoManual := "DB_R134a_BU_Values".Valve.Spare_1.Input.OpModeAutoManual, I_AutoOn := "DB_R134a_BU_Values".Valve.Spare_1.Input.AutoOn, I_AutoOff := "DB_R134a_BU_Values".Valve.Spare_1.Input.AutoOff, I_ManualOn := "DB_R134a_BU_Values".Valve.Spare_1.Input.ManualOn, I_ManualOff := "DB_R134a_BU_Values".Valve.Spare_1.Input.ManualOff, I_Release := "DB_R134a_BU_Values".Valve.Spare_1.Input.Release, I_SafetyRelease := "DB_R134a_BU_Values".Valve.Spare_1.Input.SafetyRelease, I_ID := WSTRING#'1KM1VI1KKP10KKR14', I_TextName_Language := "DB_R134a_BU_Values".Valve.Spare_1.Input.TextName_Language, I_Language := "DB_HMI_1".Language, O_ValveOutput => "DB_R134a_BU_Values".Valve.Spare_1.Output.Valve, O_ValveHMI => "DB_R134a_BU_Values".Valve.Spare_1.HMI.Valve, O_ID => "DB_R134a_BU_Values".Valve.Spare_1.HMI.ID, O_TextName => "DB_R134a_BU_Values".Valve.Spare_1.HMI.TextName, O_Status => "DB_R134a_BU_Values".Valve.Spare_1.HMI.Status)
      Contact( "DB_R134a_BU_Values".Valve.Spare_1.Output.Valve )
      Coil( "1KM1VI1KKP10KKR14" )
   END_RUNG
   // the same network as SCL:
   #Valve_Spare_1(I_OpModeOutput := "DB_R134a_BU_Values".Valve.Spare_1.Input.OpModeOutput,   // "FB_VALVE"
                  I_OpModeAutoManual := "DB_R134a_BU_Values".Valve.Spare_1.Input.OpModeAutoManual,
                  I_AutoOn := "DB_R134a_BU_Values".Valve.Spare_1.Input.AutoOn,
                  I_AutoOff := "DB_R134a_BU_Values".Valve.Spare_1.Input.AutoOff,
                  I_ManualOn := "DB_R134a_BU_Values".Valve.Spare_1.Input.ManualOn,
                  I_ManualOff := "DB_R134a_BU_Values".Valve.Spare_1.Input.ManualOff,
                  I_Release := "DB_R134a_BU_Values".Valve.Spare_1.Input.Release,
                  I_SafetyRelease := "DB_R134a_BU_Values".Valve.Spare_1.Input.SafetyRelease,
                  I_ID := WSTRING#'1KM1VI1KKP10KKR14',
                  I_TextName_Language := "DB_R134a_BU_Values".Valve.Spare_1.Input.TextName_Language,
                  I_Language := "DB_HMI_1".Language,
                  O_ValveOutput => "DB_R134a_BU_Values".Valve.Spare_1.Output.Valve,
                  O_ValveHMI => "DB_R134a_BU_Values".Valve.Spare_1.HMI.Valve,
                  O_ID => "DB_R134a_BU_Values".Valve.Spare_1.HMI.ID,
                  O_TextName => "DB_R134a_BU_Values".Valve.Spare_1.HMI.TextName,
                  O_Status => "DB_R134a_BU_Values".Valve.Spare_1.HMI.Status,
                  ENO => #_w1);
   "1KM1VI1KKP10KKR14" := #_w1 AND "DB_R134a_BU_Values".Valve.Spare_1.Output.Valve;
END_REGION

REGION Network 35: [Spare_2] valve logic
   // Setup  //  Parametrierungshinweise
   // I_OpModeOutput  -->
   // 0=I_AutoOn schaltet den Ausgang Ein und Aus; 1=I_AutoOn schaltet ein und I_AutoAus schaltet aus
   // 0=I_AutoOn switches on and off; 1=I_AutoOn switches on and I_AutoOff switches off
   // 
   // I_OpModeAutoManual -->
   // 0=Automatik; 1=Hand
   // 0=Automatic; 1=Manual
   // 
   // I_AutoOn -->
   // 1=Automatik Ein, Eingang für die normalen Ventilverschaltungsbedingungen
   // 1=Automatic On, Input for the normal valve conditions
   // 
   // I_Release -->
   // 1=Freigabe, Eingang für die Fehlerbedingungen
   // 1=Release, Input for fault conditions
   // 
   // I_SafetyRelease -->
   // 1=Sicherheitsfreigabe, Eingang für zusätzliche Schaltbefehle aus dem Sicherheitsprogramm
   // 1=Safety release, Input for additional safety conditions from the safety program
   RUNG wire#powerrail
      Move(in := 0, out1 => "DB_R134a_BU_Values".Valve.Spare_2.Input.OpModeOutput)
      Move(in := "DB_R134a_AT_2_Values".OperationMode.ManualValveControl, out1 => "DB_R134a_BU_Values".Valve.Spare_2.Input.OpModeAutoManual)
      { S7_Templates := "SrcType := Int" } EQ_Contact(in1 := "DB_R134a_BU_Values".Valve.Spare_2.Input.OpModeAutoManual, in2 := 0)
      R_Coil( "DB_R134a_BU_Values".Valve.Spare_2.Input.ManualOn )
   END_RUNG
   RUNG wire#powerrail
      Contact( #Tmp_EnableOperation )
      Contact( "AlwaysFALSE" )
      Coil( "DB_R134a_BU_Values".Valve.Spare_2.Input.AutoOn )
   END_RUNG
   RUNG wire#powerrail
      Coil( "DB_R134a_BU_Values".Valve.Spare_2.Input.Release )
   END_RUNG
   RUNG wire#powerrail
      Coil( "DB_R134a_BU_Values".Valve.Spare_2.Input.SafetyRelease )
   END_RUNG
   RUNG wire#powerrail
      MOVE_BLK_VARIANT(SRC := "DB_R134a_1_StepData".Valve[1].Language, COUNT := 4, SRC_INDEX := 0, DEST_INDEX := 0, Ret_Val => #Tmp_ReturnValue, DEST => "DB_R134a_BU_Values".Valve.Spare_2.Input.TextName_Language)
   END_RUNG
   // the same network as SCL:
   "DB_R134a_BU_Values".Valve.Spare_2.Input.OpModeOutput := 0;
   "DB_R134a_BU_Values".Valve.Spare_2.Input.OpModeAutoManual := "DB_R134a_AT_2_Values".OperationMode.ManualValveControl;
   IF "DB_R134a_BU_Values".Valve.Spare_2.Input.OpModeAutoManual = 0 THEN
       "DB_R134a_BU_Values".Valve.Spare_2.Input.ManualOn := FALSE;
   END_IF;
   "DB_R134a_BU_Values".Valve.Spare_2.Input.AutoOn := #Tmp_EnableOperation AND "AlwaysFALSE";
   "DB_R134a_BU_Values".Valve.Spare_2.Input.Release := TRUE;
   "DB_R134a_BU_Values".Valve.Spare_2.Input.SafetyRelease := TRUE;
   #Tmp_ReturnValue := MOVE_BLK_VARIANT(SRC := "DB_R134a_1_StepData".Valve[1].Language,
                           COUNT := 4,
                           SRC_INDEX := 0,
                           DEST_INDEX := 0,
                           DEST => "DB_R134a_BU_Values".Valve.Spare_2.Input.TextName_Language);
END_REGION

REGION Network 36: [Spare_2] valve 1KM1VI1KKP10KKR12 - xxx.. - spare // Reserve
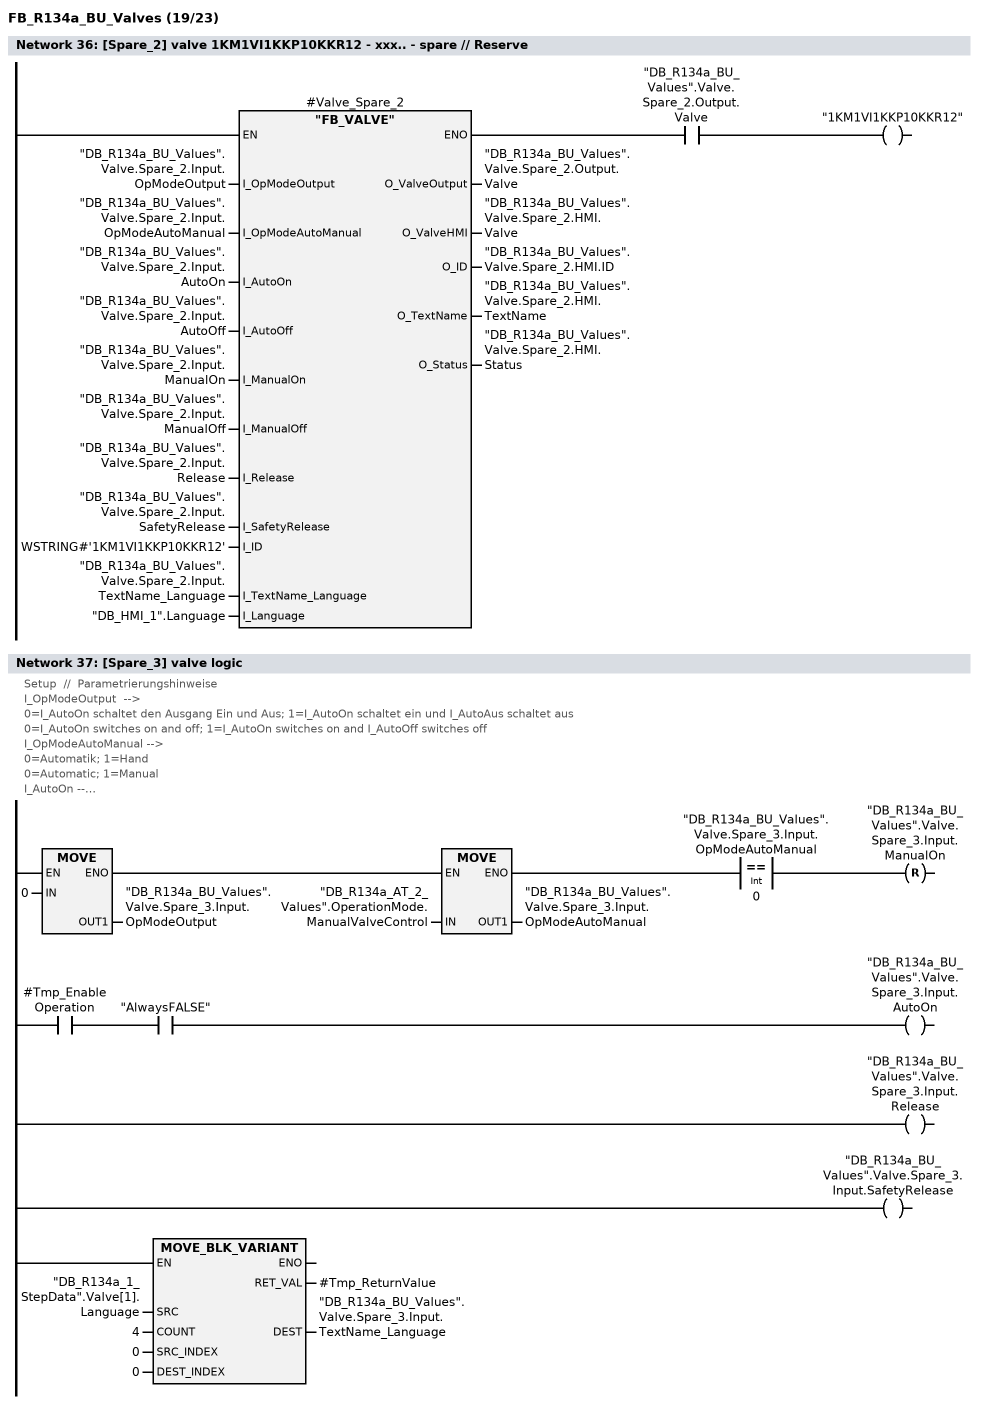
   RUNG wire#powerrail
      #Valve_Spare_2(I_OpModeOutput := "DB_R134a_BU_Values".Valve.Spare_2.Input.OpModeOutput, I_OpModeAutoManual := "DB_R134a_BU_Values".Valve.Spare_2.Input.OpModeAutoManual, I_AutoOn := "DB_R134a_BU_Values".Valve.Spare_2.Input.AutoOn, I_AutoOff := "DB_R134a_BU_Values".Valve.Spare_2.Input.AutoOff, I_ManualOn := "DB_R134a_BU_Values".Valve.Spare_2.Input.ManualOn, I_ManualOff := "DB_R134a_BU_Values".Valve.Spare_2.Input.ManualOff, I_Release := "DB_R134a_BU_Values".Valve.Spare_2.Input.Release, I_SafetyRelease := "DB_R134a_BU_Values".Valve.Spare_2.Input.SafetyRelease, I_ID := WSTRING#'1KM1VI1KKP10KKR12', I_TextName_Language := "DB_R134a_BU_Values".Valve.Spare_2.Input.TextName_Language, I_Language := "DB_HMI_1".Language, O_ValveOutput => "DB_R134a_BU_Values".Valve.Spare_2.Output.Valve, O_ValveHMI => "DB_R134a_BU_Values".Valve.Spare_2.HMI.Valve, O_ID => "DB_R134a_BU_Values".Valve.Spare_2.HMI.ID, O_TextName => "DB_R134a_BU_Values".Valve.Spare_2.HMI.TextName, O_Status => "DB_R134a_BU_Values".Valve.Spare_2.HMI.Status)
      Contact( "DB_R134a_BU_Values".Valve.Spare_2.Output.Valve )
      Coil( "1KM1VI1KKP10KKR12" )
   END_RUNG
   // the same network as SCL:
   #Valve_Spare_2(I_OpModeOutput := "DB_R134a_BU_Values".Valve.Spare_2.Input.OpModeOutput,   // "FB_VALVE"
                  I_OpModeAutoManual := "DB_R134a_BU_Values".Valve.Spare_2.Input.OpModeAutoManual,
                  I_AutoOn := "DB_R134a_BU_Values".Valve.Spare_2.Input.AutoOn,
                  I_AutoOff := "DB_R134a_BU_Values".Valve.Spare_2.Input.AutoOff,
                  I_ManualOn := "DB_R134a_BU_Values".Valve.Spare_2.Input.ManualOn,
                  I_ManualOff := "DB_R134a_BU_Values".Valve.Spare_2.Input.ManualOff,
                  I_Release := "DB_R134a_BU_Values".Valve.Spare_2.Input.Release,
                  I_SafetyRelease := "DB_R134a_BU_Values".Valve.Spare_2.Input.SafetyRelease,
                  I_ID := WSTRING#'1KM1VI1KKP10KKR12',
                  I_TextName_Language := "DB_R134a_BU_Values".Valve.Spare_2.Input.TextName_Language,
                  I_Language := "DB_HMI_1".Language,
                  O_ValveOutput => "DB_R134a_BU_Values".Valve.Spare_2.Output.Valve,
                  O_ValveHMI => "DB_R134a_BU_Values".Valve.Spare_2.HMI.Valve,
                  O_ID => "DB_R134a_BU_Values".Valve.Spare_2.HMI.ID,
                  O_TextName => "DB_R134a_BU_Values".Valve.Spare_2.HMI.TextName,
                  O_Status => "DB_R134a_BU_Values".Valve.Spare_2.HMI.Status,
                  ENO => #_w1);
   "1KM1VI1KKP10KKR12" := #_w1 AND "DB_R134a_BU_Values".Valve.Spare_2.Output.Valve;
END_REGION

